LIN {X 0,Y 220.95,Z 365.337,A -85,B 0,C 180,E1 -21122.312,E2 -21122.312} C_VEL
LIN {X 0,Y 219.711,Z 400.675,A -85,B 0,C 180,E1 -21123.481,E2 -21123.481} C_VEL
LIN {X 0,Y 218.85,Z 411.091,A -85,B 0,C 180,E1 -21124.077,E2 -21124.077} C_VEL
LIN {X 0,Y 217.457,Z 422.982,A -85,B 0,C 180,E1 -21125.157,E2 -21125.157} C_VEL
LIN {X 0,Y 216.121,Z 431.792,A -85,B 0,C 180,E1 -21126.271,E2 -21126.271} C_VEL
LIN {X 0,Y 214.526,Z 440.18,A -85,B 0,C 180,E1 -21127.615,E2 -21127.615} C_VEL
LIN {X 0,Y 212.777,Z 448.104,A -85,B 0,C 180,E1 -21129.203,E2 -21129.203} C_VEL
LIN {X 0,Y 210.956,Z 455.495,A -85,B 0,C 180,E1 -21131.046,E2 -21131.046} C_VEL
LIN {X 0,Y 209.085,Z 462.983,A -85,B 0,C 180,E1 -21133.399,E2 -21133.399} C_VEL
LIN {X 0,Y 207.25,Z 469.848,A -85,B 0,C 180,E1 -21136.269,E2 -21136.269} C_VEL
LIN {X 0,Y 205.923,Z 475.039,A -85,B 0,C 180,E1 -21139.181,E2 -21139.181} C_VEL
LIN {X 0,Y 205.254,Z 477.703,A -85,B 0,C 180,E1 -21141.137,E2 -21141.137} C_VEL
LIN {X 0,Y 204.593,Z 480.62,A -85,B 0,C 180,E1 -21144.085,E2 -21144.085} C_VEL
LIN {X 0,Y 204.405,Z 481.892,A -85,B 0,C 180,E1 -21146.057,E2 -21146.057} C_VEL
LIN {X 0,Y 204.322,Z 482.694,A -85,B 0,C 180,E1 -21148.029,E2 -21148.029} C_VEL
LIN {X 0,Y 204.302,Z 482.999,A -85,B 0,C 180,E1 -21150,E2 -21150} C_VEL
LIN {X 0,Y 204.315,Z 482.717,A -85,B 0,C 180,E1 -21151.971,E2 -21151.971} C_VEL
LIN {X 0,Y 204.439,Z 481.698,A -85,B 0,C 180,E1 -21154.487,E2 -21154.487} C_VEL
LIN {X 0,Y 204.992,Z 479.021,A -85,B 0,C 180,E1 -21157.882,E2 -21157.882} C_VEL
LIN {X 0,Y 205.895,Z 475.26,A -85,B 0,C 180,E1 -21160.82,E2 -21160.82} C_VEL
LIN {X 0,Y 207.184,Z 470.127,A -85,B 0,C 180,E1 -21163.736,E2 -21163.736} C_VEL
LIN {X 0,Y 208.712,Z 464.607,A -85,B 0,C 180,E1 -21166.129,E2 -21166.129} C_VEL
LIN {X 0,Y 210.499,Z 457.67,A -85,B 0,C 180,E1 -21168.492,E2 -21168.492} C_VEL
LIN {X 0,Y 212.455,Z 449.707,A -85,B 0,C 180,E1 -21170.577,E2 -21170.577} C_VEL
LIN {X 0,Y 214.197,Z 442.115,A -85,B 0,C 180,E1 -21172.168,E2 -21172.168} C_VEL
LIN {X 0,Y 215.813,Z 434.156,A -85,B 0,C 180,E1 -21173.51,E2 -21173.51} C_VEL
LIN {X 0,Y 216.859,Z 427.803,A -85,B 0,C 180,E1 -21174.406,E2 -21174.406} C_VEL
LIN {X 0,Y 218.133,Z 418.906,A -85,B 0,C 180,E1 -21175.386,E2 -21175.386} C_VEL
LIN {X 0,Y 219.062,Z 409.592,A -85,B 0,C 180,E1 -21176.159,E2 -21176.159} C_VEL
LIN {X 0,Y 219.757,Z 400.653,A -85,B 0,C 180,E1 -21176.661,E2 -21176.661} C_VEL
LIN {X 0,Y 221.039,Z 365.121,A -85,B 0,C 180,E1 -21177.832,E2 -21177.832} C_VEL
LIN {X 0,Y 218.467,Z 349.485,A -85,B 0,C 180,E1 -21178.761,E2 -21178.761} C_VEL
LIN {X 0,Y 212.436,Z 334.283,A -85,B 0,C 180,E1 -21180.238,E2 -21180.238} C_VEL
LIN {X 0,Y 207.752,Z 323.941,A -85,B 0,C 180,E1 -21181.473,E2 -21181.473} C_VEL
LIN {X 0,Y 207.162,Z 321.361,A -85,B 0,C 180,E1 -21182.874,E2 -21182.874} C_VEL
LIN {X 0,Y 206.738,Z 319.61,A -85,B 0,C 180,E1 -21184.118,E2 -21184.118} C_VEL
LIN {X 0,Y 206.671,Z 319.549,A -85,B 0,C 180,E1 -21188.543,E2 -21188.543} C_VEL
LIN {X 0,Y 206.616,Z 319.531,A -85,B 0,C 180,E1 -21192.866,E2 -21192.866} C_VEL
LIN {X 0,Y 206.615,Z 319.554,A -85,B 0,C 180,E1 -21197.133,E2 -21197.133} C_VEL
LIN {X 0,Y 206.659,Z 319.506,A -85,B 0,C 180,E1 -21202.255,E2 -21202.255} C_VEL
LIN {X 0,Y 206.697,Z 319.538,A -85,B 0,C 180,E1 -21204.688,E2 -21204.688} C_VEL
LIN {X 0,Y 206.691,Z 319.539,A -85,B 0,C 180,E1 -21209.333,E2 -21209.333} C_VEL
LIN {X 0,Y 206.682,Z 319.552,A -85,B 0,C 180,E1 -21213.765,E2 -21213.765} C_VEL
LIN {X 0,Y 206.707,Z 319.528,A -85,B 0,C 180,E1 -21218.037,E2 -21218.037} C_VEL
LIN {X 0,Y 206.799,Z 319.538,A -85,B 0,C 180,E1 -21222.19,E2 -21222.19} C_VEL
LIN {X 0,Y 206.846,Z 319.508,A -85,B 0,C 180,E1 -21226.241,E2 -21226.241} C_VEL
LIN {X 0,Y 207.073,Z 319.503,A -85,B 0,C 180,E1 -21230.229,E2 -21230.229} C_VEL
LIN {X 0,Y 207.03,Z 319.487,A -85,B 0,C 180,E1 -21234.155,E2 -21234.155} C_VEL
LIN {X 0,Y 207.336,Z 319.463,A -85,B 0,C 180,E1 -21238.057,E2 -21238.057} C_VEL
LIN {X 0,Y 207.473,Z 319.455,A -85,B 0,C 180,E1 -21240,E2 -21240} C_VEL
LIN {X 0,Y 207.333,Z 319.464,A -85,B 0,C 180,E1 -21241.942,E2 -21241.942} C_VEL
LIN {X 0,Y 207.111,Z 319.493,A -85,B 0,C 180,E1 -21247.801,E2 -21247.801} C_VEL
LIN {X 0,Y 206.896,Z 319.513,A -85,B 0,C 180,E1 -21251.76,E2 -21251.76} C_VEL
LIN {X 0,Y 206.794,Z 319.527,A -85,B 0,C 180,E1 -21255.776,E2 -21255.776} C_VEL
LIN {X 0,Y 206.705,Z 319.542,A -85,B 0,C 180,E1 -21259.877,E2 -21259.877} C_VEL
LIN {X 0,Y 206.716,Z 319.539,A -85,B 0,C 180,E1 -21264.078,E2 -21264.078} C_VEL
LIN {X 0,Y 206.682,Z 319.541,A -85,B 0,C 180,E1 -21268.428,E2 -21268.428} C_VEL
LIN {X 0,Y 206.69,Z 319.552,A -85,B 0,C 180,E1 -21272.959,E2 -21272.959} C_VEL
LIN {X 0,Y 206.662,Z 319.507,A -85,B 0,C 180,E1 -21277.743,E2 -21277.743} C_VEL
LIN {X 0,Y 206.627,Z 319.53,A -85,B 0,C 180,E1 -21281.559,E2 -21281.559} C_VEL
LIN {X 0,Y 206.626,Z 319.552,A -85,B 0,C 180,E1 -21285.584,E2 -21285.584} C_VEL
LIN {X 0,Y 206.644,Z 319.525,A -85,B 0,C 180,E1 -21289.746,E2 -21289.746} C_VEL
LIN {X 0,Y 206.697,Z 319.53,A -85,B 0,C 180,E1 -21294.689,E2 -21294.689} C_VEL
LIN {X 0,Y 206.763,Z 319.832,A -85,B 0,C 180,E1 -21296.18,E2 -21296.18} C_VEL
LIN {X 0,Y 207.225,Z 321.798,A -85,B 0,C 180,E1 -21297.441,E2 -21297.441} C_VEL
LIN {X 0,Y 207.769,Z 324.004,A -85,B 0,C 180,E1 -21298.251,E2 -21298.251} C_VEL
LIN {X 0,Y 208.558,Z 327.091,A -85,B 0,C 180,E1 -21298.81,E2 -21298.81} C_VEL
LIN {X 0,Y 209.749,Z 332.596,A -85,B 0,C 180,E1 -21299.313,E2 -21299.313} C_VEL
LIN {X 0,Y 211.186,Z 347.134,A -85,B 0,C 180,E1 -21300.1,E2 -21300.1} C_VEL
LIN {X 0,Y 212.232,Z 351.094,A -85,B 0,C 180,E1 -21300.418,E2 -21300.418} C_VEL
LIN {X 0,Y 213.675,Z 358.475,A -85,B 0,C 180,E1 -21300.917,E2 -21300.917} C_VEL
LIN {X 0,Y 214.812,Z 367.699,A -85,B 0,C 180,E1 -21301.43,E2 -21301.43} C_VEL
LIN {X 0,Y 213.518,Z 400.025,A -85,B 0,C 180,E1 -21302.509,E2 -21302.509} C_VEL
LIN {X 0,Y 212.78,Z 409.431,A -85,B 0,C 180,E1 -21303.041,E2 -21303.041} C_VEL
LIN {X 0,Y 211.677,Z 418.832,A -85,B 0,C 180,E1 -21303.82,E2 -21303.82} C_VEL
LIN {X 0,Y 210.186,Z 429.315,A -85,B 0,C 180,E1 -21305.031,E2 -21305.031} C_VEL
LIN {X 0,Y 208.163,Z 439.443,A -85,B 0,C 180,E1 -21306.628,E2 -21306.628} C_VEL
LIN {X 0,Y 206.357,Z 447.487,A -85,B 0,C 180,E1 -21308.262,E2 -21308.262} C_VEL
LIN {X 0,Y 204.685,Z 454.131,A -85,B 0,C 180,E1 -21309.919,E2 -21309.919} C_VEL
LIN {X 0,Y 202.959,Z 460.438,A -85,B 0,C 180,E1 -21311.842,E2 -21311.842} C_VEL
LIN {X 0,Y 201.558,Z 465.676,A -85,B 0,C 180,E1 -21313.803,E2 -21313.803} C_VEL
LIN {X 0,Y 200.308,Z 470.043,A -85,B 0,C 180,E1 -21315.783,E2 -21315.783} C_VEL
LIN {X 0,Y 198.917,Z 475.192,A -85,B 0,C 180,E1 -21318.795,E2 -21318.795} C_VEL
LIN {X 0,Y 197.976,Z 478.97,A -85,B 0,C 180,E1 -21321.837,E2 -21321.837} C_VEL
LIN {X 0,Y 197.59,Z 480.702,A -85,B 0,C 180,E1 -21323.875,E2 -21323.875} C_VEL
LIN {X 0,Y 197.332,Z 481.941,A -85,B 0,C 180,E1 -21325.915,E2 -21325.915} C_VEL
LIN {X 0,Y 197.234,Z 482.71,A -85,B 0,C 180,E1 -21327.958,E2 -21327.958} C_VEL
LIN {X 0,Y 197.21,Z 483,A -85,B 0,C 180,E1 -21330,E2 -21330} C_VEL
LIN {X 0,Y 197.232,Z 482.701,A -85,B 0,C 180,E1 -21332.042,E2 -21332.042} C_VEL
LIN {X 0,Y 197.336,Z 481.816,A -85,B 0,C 180,E1 -21334.291,E2 -21334.291} C_VEL
LIN {X 0,Y 197.523,Z 480.656,A -85,B 0,C 180,E1 -21336.127,E2 -21336.127} C_VEL
LIN {X 0,Y 198.238,Z 477.754,A -85,B 0,C 180,E1 -21339.18,E2 -21339.18} C_VEL
LIN {X 0,Y 198.911,Z 475.107,A -85,B 0,C 180,E1 -21341.205,E2 -21341.205} C_VEL
LIN {X 0,Y 200.301,Z 469.932,A -85,B 0,C 180,E1 -21344.218,E2 -21344.218} C_VEL
LIN {X 0,Y 202.263,Z 463.105,A -85,B 0,C 180,E1 -21347.178,E2 -21347.178} C_VEL
LIN {X 0,Y 204.226,Z 455.644,A -85,B 0,C 180,E1 -21349.604,E2 -21349.604} C_VEL
LIN {X 0,Y 206.112,Z 448.282,A -85,B 0,C 180,E1 -21351.503,E2 -21351.503} C_VEL
LIN {X 0,Y 207.939,Z 440.395,A -85,B 0,C 180,E1 -21353.135,E2 -21353.135} C_VEL
LIN {X 0,Y 209.55,Z 432.053,A -85,B 0,C 180,E1 -21354.521,E2 -21354.521} C_VEL
LIN {X 0,Y 211.157,Z 422.131,A -85,B 0,C 180,E1 -21355.803,E2 -21355.803} C_VEL
LIN {X 0,Y 212.607,Z 410.515,A -85,B 0,C 180,E1 -21356.836,E2 -21356.836} C_VEL
LIN {X 0,Y 213.421,Z 400.836,A -85,B 0,C 180,E1 -21357.402,E2 -21357.402} C_VEL
LIN {X 0,Y 214.677,Z 366.325,A -85,B 0,C 180,E1 -21358.58,E2 -21358.58} C_VEL
LIN {X 0,Y 212.372,Z 351.475,A -85,B 0,C 180,E1 -21359.482,E2 -21359.482} C_VEL
LIN {X 0,Y 206.305,Z 336.552,A -85,B 0,C 180,E1 -21361.03,E2 -21361.03} C_VEL
LIN {X 0,Y 200.492,Z 323.95,A -85,B 0,C 180,E1 -21362.63,E2 -21362.63} C_VEL
LIN {X 0,Y 199.816,Z 321.165,A -85,B 0,C 180,E1 -21364.246,E2 -21364.246} C_VEL
LIN {X 0,Y 199.669,Z 320.48,A -85,B 0,C 180,E1 -21364.845,E2 -21364.845} C_VEL
LIN {X 0,Y 199.593,Z 320.412,A -85,B 0,C 180,E1 -21369.331,E2 -21369.331} C_VEL
LIN {X 0,Y 199.562,Z 320.404,A -85,B 0,C 180,E1 -21372.306,E2 -21372.306} C_VEL
LIN {X 0,Y 199.572,Z 320.438,A -85,B 0,C 180,E1 -21375.227,E2 -21375.227} C_VEL
LIN {X 0,Y 199.566,Z 320.413,A -85,B 0,C 180,E1 -21378.002,E2 -21378.002} C_VEL
LIN {X 0,Y 199.593,Z 320.378,A -85,B 0,C 180,E1 -21380.772,E2 -21380.772} C_VEL
LIN {X 0,Y 199.607,Z 320.432,A -85,B 0,C 180,E1 -21385.713,E2 -21385.713} C_VEL
LIN {X 0,Y 199.681,Z 320.42,A -85,B 0,C 180,E1 -21388.134,E2 -21388.134} C_VEL
LIN {X 0,Y 199.63,Z 320.428,A -85,B 0,C 180,E1 -21392.764,E2 -21392.764} C_VEL
LIN {X 0,Y 199.666,Z 320.405,A -85,B 0,C 180,E1 -21397.221,E2 -21397.221} C_VEL
LIN {X 0,Y 199.741,Z 320.416,A -85,B 0,C 180,E1 -21401.803,E2 -21401.803} C_VEL
LIN {X 0,Y 199.763,Z 320.39,A -85,B 0,C 180,E1 -21405.743,E2 -21405.743} C_VEL
LIN {X 0,Y 200.019,Z 320.379,A -85,B 0,C 180,E1 -21409.882,E2 -21409.882} C_VEL
LIN {X 0,Y 199.994,Z 320.363,A -85,B 0,C 180,E1 -21413.949,E2 -21413.949} C_VEL
LIN {X 0,Y 200.278,Z 320.342,A -85,B 0,C 180,E1 -21417.989,E2 -21417.989} C_VEL
LIN {X 0,Y 200.44,Z 320.331,A -85,B 0,C 180,E1 -21420,E2 -21420} C_VEL
LIN {X 0,Y 199.973,Z 320.362,A -85,B 0,C 180,E1 -21424.031,E2 -21424.031} C_VEL
LIN {X 0,Y 200.06,Z 320.373,A -85,B 0,C 180,E1 -21428.078,E2 -21428.078} C_VEL
LIN {X 0,Y 199.846,Z 320.388,A -85,B 0,C 180,E1 -21432.181,E2 -21432.181} C_VEL
LIN {X 0,Y 199.735,Z 320.41,A -85,B 0,C 180,E1 -21436.35,E2 -21436.35} C_VEL
LIN {X 0,Y 199.639,Z 320.417,A -85,B 0,C 180,E1 -21440.612,E2 -21440.612} C_VEL
LIN {X 0,Y 199.631,Z 320.427,A -85,B 0,C 180,E1 -21444.99,E2 -21444.99} C_VEL
LIN {X 0,Y 199.604,Z 320.416,A -85,B 0,C 180,E1 -21449.534,E2 -21449.534} C_VEL
LIN {X 0,Y 199.662,Z 320.425,A -85,B 0,C 180,E1 -21452.353,E2 -21452.353} C_VEL
LIN {X 0,Y 199.613,Z 320.397,A -85,B 0,C 180,E1 -21456.765,E2 -21456.765} C_VEL
LIN {X 0,Y 199.591,Z 320.379,A -85,B 0,C 180,E1 -21459.332,E2 -21459.332} C_VEL
LIN {X 0,Y 199.563,Z 320.418,A -85,B 0,C 180,E1 -21462.308,E2 -21462.308} C_VEL
LIN {X 0,Y 199.573,Z 320.435,A -85,B 0,C 180,E1 -21465.228,E2 -21465.228} C_VEL
LIN {X 0,Y 199.567,Z 320.401,A -85,B 0,C 180,E1 -21468.003,E2 -21468.003} C_VEL
LIN {X 0,Y 199.596,Z 320.412,A -85,B 0,C 180,E1 -21470.773,E2 -21470.773} C_VEL
LIN {X 0,Y 199.728,Z 320.655,A -85,B 0,C 180,E1 -21475.453,E2 -21475.453} C_VEL
LIN {X 0,Y 200.467,Z 323.816,A -85,B 0,C 180,E1 -21477.38,E2 -21477.38} C_VEL
LIN {X 0,Y 202.785,Z 329.044,A -85,B 0,C 180,E1 -21478.109,E2 -21478.109} C_VEL
LIN {X 0,Y 208.66,Z 342.11,A -85,B 0,C 180,E1 -21479.62,E2 -21479.62} C_VEL
LIN {X 0,Y 212.507,Z 352.019,A -85,B 0,C 180,E1 -21480.604,E2 -21480.604} C_VEL
LIN {X 0,Y 214.697,Z 366.722,A -85,B 0,C 180,E1 -21481.483,E2 -21481.483} C_VEL
LIN {X 0,Y 213.422,Z 400.147,A -85,B 0,C 180,E1 -21482.608,E2 -21482.608} C_VEL
LIN {X 0,Y 212.631,Z 409.776,A -85,B 0,C 180,E1 -21483.153,E2 -21483.153} C_VEL
LIN {X 0,Y 211.516,Z 419.764,A -85,B 0,C 180,E1 -21484.006,E2 -21484.006} C_VEL
LIN {X 0,Y 209.91,Z 430.293,A -85,B 0,C 180,E1 -21485.26,E2 -21485.26} C_VEL
LIN {X 0,Y 207.983,Z 440.184,A -85,B 0,C 180,E1 -21486.87,E2 -21486.87} C_VEL
LIN {X 0,Y 206.16,Z 448.107,A -85,B 0,C 180,E1 -21488.503,E2 -21488.503} C_VEL
LIN {X 0,Y 204.262,Z 455.497,A -85,B 0,C 180,E1 -21490.4,E2 -21490.4} C_VEL
LIN {X 0,Y 202.29,Z 462.985,A -85,B 0,C 180,E1 -21492.824,E2 -21492.824} C_VEL
LIN {X 0,Y 200.342,Z 469.849,A -85,B 0,C 180,E1 -21495.785,E2 -21495.785} C_VEL
LIN {X 0,Y 198.94,Z 475.04,A -85,B 0,C 180,E1 -21498.796,E2 -21498.796} C_VEL
LIN {X 0,Y 198.242,Z 477.703,A -85,B 0,C 180,E1 -21500.82,E2 -21500.82} C_VEL
LIN {X 0,Y 197.525,Z 480.621,A -85,B 0,C 180,E1 -21503.873,E2 -21503.873} C_VEL
LIN {X 0,Y 197.326,Z 481.893,A -85,B 0,C 180,E1 -21505.915,E2 -21505.915} C_VEL
LIN {X 0,Y 197.234,Z 482.694,A -85,B 0,C 180,E1 -21507.958,E2 -21507.958} C_VEL
LIN {X 0,Y 197.211,Z 482.999,A -85,B 0,C 180,E1 -21510,E2 -21510} C_VEL
LIN {X 0,Y 197.228,Z 482.717,A -85,B 0,C 180,E1 -21512.042,E2 -21512.042} C_VEL
LIN {X 0,Y 197.338,Z 481.865,A -85,B 0,C 180,E1 -21514.291,E2 -21514.291} C_VEL
LIN {X 0,Y 197.525,Z 480.738,A -85,B 0,C 180,E1 -21516.127,E2 -21516.127} C_VEL
LIN {X 0,Y 198.239,Z 477.869,A -85,B 0,C 180,E1 -21519.18,E2 -21519.18} C_VEL
LIN {X 0,Y 198.907,Z 475.258,A -85,B 0,C 180,E1 -21521.205,E2 -21521.205} C_VEL
LIN {X 0,Y 200.282,Z 470.126,A -85,B 0,C 180,E1 -21524.219,E2 -21524.219} C_VEL
LIN {X 0,Y 201.894,Z 464.605,A -85,B 0,C 180,E1 -21526.689,E2 -21526.689} C_VEL
LIN {X 0,Y 203.756,Z 457.667,A -85,B 0,C 180,E1 -21529.127,E2 -21529.127} C_VEL
LIN {X 0,Y 205.831,Z 449.703,A -85,B 0,C 180,E1 -21531.271,E2 -21531.271} C_VEL
LIN {X 0,Y 207.639,Z 442.111,A -85,B 0,C 180,E1 -21532.907,E2 -21532.907} C_VEL
LIN {X 0,Y 209.328,Z 434.151,A -85,B 0,C 180,E1 -21534.285,E2 -21534.285} C_VEL
LIN {X 0,Y 210.745,Z 425.924,A -85,B 0,C 180,E1 -21535.426,E2 -21535.426} C_VEL
LIN {X 0,Y 211.861,Z 417.634,A -85,B 0,C 180,E1 -21536.332,E2 -21536.332} C_VEL
LIN {X 0,Y 212.757,Z 409.338,A -85,B 0,C 180,E1 -21537.015,E2 -21537.015} C_VEL
LIN {X 0,Y 213.439,Z 400.806,A -85,B 0,C 180,E1 -21537.507,E2 -21537.507} C_VEL
LIN {X 0,Y 214.789,Z 366.132,A -85,B 0,C 180,E1 -21538.677,E2 -21538.677} C_VEL
LIN {X 0,Y 212.416,Z 351.696,A -85,B 0,C 180,E1 -21539.576,E2 -21539.576} C_VEL
LIN {X 0,Y 206.152,Z 336.12,A -85,B 0,C 180,E1 -21541.187,E2 -21541.187} C_VEL
LIN {X 0,Y 200.525,Z 323.991,A -85,B 0,C 180,E1 -21542.737,E2 -21542.737} C_VEL
LIN {X 0,Y 200.187,Z 322.632,A -85,B 0,C 180,E1 -21543.385,E2 -21543.385} C_VEL
LIN {X 0,Y 199.67,Z 320.525,A -85,B 0,C 180,E1 -21544.844,E2 -21544.844} C_VEL
LIN {X 0,Y 199.593,Z 320.414,A -85,B 0,C 180,E1 -21549.331,E2 -21549.331} C_VEL
LIN {X 0,Y 199.563,Z 320.403,A -85,B 0,C 180,E1 -21552.306,E2 -21552.306} C_VEL
LIN {X 0,Y 199.573,Z 320.437,A -85,B 0,C 180,E1 -21555.226,E2 -21555.226} C_VEL
LIN {X 0,Y 199.566,Z 320.416,A -85,B 0,C 180,E1 -21558.001,E2 -21558.001} C_VEL
LIN {X 0,Y 199.59,Z 320.379,A -85,B 0,C 180,E1 -21560.773,E2 -21560.773} C_VEL
LIN {X 0,Y 199.608,Z 320.43,A -85,B 0,C 180,E1 -21565.712,E2 -21565.712} C_VEL
LIN {X 0,Y 199.682,Z 320.421,A -85,B 0,C 180,E1 -21568.133,E2 -21568.133} C_VEL
LIN {X 0,Y 199.631,Z 320.427,A -85,B 0,C 180,E1 -21572.763,E2 -21572.763} C_VEL
LIN {X 0,Y 199.666,Z 320.406,A -85,B 0,C 180,E1 -21577.22,E2 -21577.22} C_VEL
LIN {X 0,Y 199.742,Z 320.416,A -85,B 0,C 180,E1 -21581.802,E2 -21581.802} C_VEL
LIN {X 0,Y 199.763,Z 320.39,A -85,B 0,C 180,E1 -21585.743,E2 -21585.743} C_VEL
LIN {X 0,Y 200.019,Z 320.379,A -85,B 0,C 180,E1 -21589.881,E2 -21589.881} C_VEL
LIN {X 0,Y 199.994,Z 320.364,A -85,B 0,C 180,E1 -21593.948,E2 -21593.948} C_VEL
LIN {X 0,Y 200.278,Z 320.341,A -85,B 0,C 180,E1 -21597.989,E2 -21597.989} C_VEL
LIN {X 0,Y 200.44,Z 320.331,A -85,B 0,C 180,E1 -21600,E2 -21600} C_VEL
LIN {X 0,Y 199.972,Z 320.362,A -85,B 0,C 180,E1 -21604.03,E2 -21604.03} C_VEL
LIN {X 0,Y 200.06,Z 320.373,A -85,B 0,C 180,E1 -21608.078,E2 -21608.078} C_VEL
LIN {X 0,Y 199.846,Z 320.388,A -85,B 0,C 180,E1 -21612.181,E2 -21612.181} C_VEL
LIN {X 0,Y 199.735,Z 320.411,A -85,B 0,C 180,E1 -21616.349,E2 -21616.349} C_VEL
LIN {X 0,Y 199.638,Z 320.416,A -85,B 0,C 180,E1 -21620.612,E2 -21620.612} C_VEL
LIN {X 0,Y 199.631,Z 320.427,A -85,B 0,C 180,E1 -21624.99,E2 -21624.99} C_VEL
LIN {X 0,Y 199.603,Z 320.416,A -85,B 0,C 180,E1 -21629.534,E2 -21629.534} C_VEL
LIN {X 0,Y 199.661,Z 320.426,A -85,B 0,C 180,E1 -21632.353,E2 -21632.353} C_VEL
LIN {X 0,Y 199.612,Z 320.395,A -85,B 0,C 180,E1 -21636.765,E2 -21636.765} C_VEL
LIN {X 0,Y 199.59,Z 320.379,A -85,B 0,C 180,E1 -21639.332,E2 -21639.332} C_VEL
LIN {X 0,Y 199.562,Z 320.421,A -85,B 0,C 180,E1 -21642.308,E2 -21642.308} C_VEL
LIN {X 0,Y 199.572,Z 320.434,A -85,B 0,C 180,E1 -21645.228,E2 -21645.228} C_VEL
LIN {X 0,Y 199.566,Z 320.401,A -85,B 0,C 180,E1 -21648.003,E2 -21648.003} C_VEL
LIN {X 0,Y 199.594,Z 320.415,A -85,B 0,C 180,E1 -21650.773,E2 -21650.773} C_VEL
LIN {X 0,Y 199.713,Z 320.637,A -85,B 0,C 180,E1 -21655.307,E2 -21655.307} C_VEL
LIN {X 0,Y 200.423,Z 323.64,A -85,B 0,C 180,E1 -21657.208,E2 -21657.208} C_VEL
LIN {X 0,Y 201.812,Z 326.976,A -85,B 0,C 180,E1 -21657.734,E2 -21657.734} C_VEL
LIN {X 0,Y 207.532,Z 339.186,A -85,B 0,C 180,E1 -21659.21,E2 -21659.21} C_VEL
LIN {X 0,Y 212.232,Z 351.094,A -85,B 0,C 180,E1 -21660.418,E2 -21660.418} C_VEL
LIN {X 0,Y 213.046,Z 354.757,A -85,B 0,C 180,E1 -21660.681,E2 -21660.681} C_VEL
LIN {X 0,Y 212.87,Z 360.592,A -85,B 0,C 180,E1 -21660.876,E2 -21660.876} C_VEL
LIN {X 0,Y 211.652,Z 366.44,A -85,B 0,C 180,E1 -21660.915,E2 -21660.915} C_VEL
LIN {X 0,Y 208.505,Z 378.509,A -85,B 0,C 180,E1 -21660.899,E2 -21660.899} C_VEL
LIN {X 0,Y 208.016,Z 382.602,A -85,B 0,C 180,E1 -21660.983,E2 -21660.983} C_VEL
LIN {X 0,Y 207.142,Z 402.34,A -85,B 0,C 180,E1 -21661.71,E2 -21661.71} C_VEL
LIN {X 0,Y 206.016,Z 413.671,A -85,B 0,C 180,E1 -21662.456,E2 -21662.456} C_VEL
LIN {X 0,Y 204.623,Z 423.738,A -85,B 0,C 180,E1 -21663.481,E2 -21663.481} C_VEL
LIN {X 0,Y 203.157,Z 432.399,A -85,B 0,C 180,E1 -21664.654,E2 -21664.654} C_VEL
LIN {X 0,Y 201.412,Z 440.676,A -85,B 0,C 180,E1 -21666.069,E2 -21666.069} C_VEL
LIN {X 0,Y 199.515,Z 448.511,A -85,B 0,C 180,E1 -21667.749,E2 -21667.749} C_VEL
LIN {X 0,Y 197.557,Z 455.837,A -85,B 0,C 180,E1 -21669.706,E2 -21669.706} C_VEL
LIN {X 0,Y 195.486,Z 463.268,A -85,B 0,C 180,E1 -21672.207,E2 -21672.207} C_VEL
LIN {X 0,Y 193.42,Z 470.044,A -85,B 0,C 180,E1 -21675.265,E2 -21675.265} C_VEL
LIN {X 0,Y 191.951,Z 475.193,A -85,B 0,C 180,E1 -21678.383,E2 -21678.383} C_VEL
LIN {X 0,Y 190.955,Z 478.971,A -85,B 0,C 180,E1 -21681.534,E2 -21681.534} C_VEL
LIN {X 0,Y 190.528,Z 480.703,A -85,B 0,C 180,E1 -21683.647,E2 -21683.647} C_VEL
LIN {X 0,Y 190.222,Z 482.043,A -85,B 0,C 180,E1 -21685.985,E2 -21685.985} C_VEL
LIN {X 0,Y 190.149,Z 482.71,A -85,B 0,C 180,E1 -21687.882,E2 -21687.882} C_VEL
LIN {X 0,Y 190.121,Z 483,A -85,B 0,C 180,E1 -21690,E2 -21690} C_VEL
LIN {X 0,Y 190.147,Z 482.701,A -85,B 0,C 180,E1 -21692.118,E2 -21692.118} C_VEL
LIN {X 0,Y 190.238,Z 481.914,A -85,B 0,C 180,E1 -21694.237,E2 -21694.237} C_VEL
LIN {X 0,Y 190.468,Z 480.656,A -85,B 0,C 180,E1 -21696.355,E2 -21696.355} C_VEL
LIN {X 0,Y 191.226,Z 477.753,A -85,B 0,C 180,E1 -21699.519,E2 -21699.519} C_VEL
LIN {X 0,Y 191.945,Z 475.105,A -85,B 0,C 180,E1 -21701.617,E2 -21701.617} C_VEL
LIN {X 0,Y 193.411,Z 469.931,A -85,B 0,C 180,E1 -21704.735,E2 -21704.735} C_VEL
LIN {X 0,Y 195.484,Z 463.103,A -85,B 0,C 180,E1 -21707.793,E2 -21707.793} C_VEL
LIN {X 0,Y 197.566,Z 455.641,A -85,B 0,C 180,E1 -21710.293,E2 -21710.293} C_VEL
LIN {X 0,Y 199.507,Z 448.279,A -85,B 0,C 180,E1 -21712.252,E2 -21712.252} C_VEL
LIN {X 0,Y 201.436,Z 440.391,A -85,B 0,C 180,E1 -21713.928,E2 -21713.928} C_VEL
LIN {X 0,Y 203.107,Z 432.048,A -85,B 0,C 180,E1 -21715.353,E2 -21715.353} C_VEL
LIN {X 0,Y 204.795,Z 422.129,A -85,B 0,C 180,E1 -21716.666,E2 -21716.666} C_VEL
LIN {X 0,Y 206.295,Z 410.586,A -85,B 0,C 180,E1 -21717.72,E2 -21717.72} C_VEL
LIN {X 0,Y 207.148,Z 401.037,A -85,B 0,C 180,E1 -21718.294,E2 -21718.294} C_VEL
LIN {X 0,Y 208.414,Z 367.129,A -85,B 0,C 180,E1 -21719.49,E2 -21719.49} C_VEL
LIN {X 0,Y 206.398,Z 353.934,A -85,B 0,C 180,E1 -21720.326,E2 -21720.326} C_VEL
LIN {X 0,Y 200.763,Z 339.948,A -85,B 0,C 180,E1 -21721.846,E2 -21721.846} C_VEL
LIN {X 0,Y 194.681,Z 327.042,A -85,B 0,C 180,E1 -21723.521,E2 -21723.521} C_VEL
LIN {X 0,Y 193.198,Z 323.808,A -85,B 0,C 180,E1 -21724.063,E2 -21724.063} C_VEL
LIN {X 0,Y 192.591,Z 321.4,A -85,B 0,C 180,E1 -21725.635,E2 -21725.635} C_VEL
LIN {X 0,Y 192.502,Z 321.285,A -85,B 0,C 180,E1 -21729.944,E2 -21729.944} C_VEL
LIN {X 0,Y 192.483,Z 321.305,A -85,B 0,C 180,E1 -21733.925,E2 -21733.925} C_VEL
LIN {X 0,Y 192.5,Z 321.273,A -85,B 0,C 180,E1 -21738.916,E2 -21738.916} C_VEL
LIN {X 0,Y 192.578,Z 321.272,A -85,B 0,C 180,E1 -21743.404,E2 -21743.404} C_VEL
LIN {X 0,Y 192.601,Z 321.307,A -85,B 0,C 180,E1 -21747.061,E2 -21747.061} C_VEL
LIN {X 0,Y 192.615,Z 321.293,A -85,B 0,C 180,E1 -21751.684,E2 -21751.684} C_VEL
LIN {X 0,Y 192.657,Z 321.283,A -85,B 0,C 180,E1 -21756.343,E2 -21756.343} C_VEL
LIN {X 0,Y 192.69,Z 321.294,A -85,B 0,C 180,E1 -21761.492,E2 -21761.492} C_VEL
LIN {X 0,Y 192.768,Z 321.264,A -85,B 0,C 180,E1 -21767.365,E2 -21767.365} C_VEL
LIN {X 0,Y 193.02,Z 321.253,A -85,B 0,C 180,E1 -21771.626,E2 -21771.626} C_VEL
LIN {X 0,Y 193.222,Z 321.22,A -85,B 0,C 180,E1 -21777.916,E2 -21777.916} C_VEL
LIN {X 0,Y 193.407,Z 321.208,A -85,B 0,C 180,E1 -21780,E2 -21780} C_VEL
LIN {X 0,Y 192.92,Z 321.238,A -85,B 0,C 180,E1 -21784.178,E2 -21784.178} C_VEL
LIN {X 0,Y 193.013,Z 321.253,A -85,B 0,C 180,E1 -21788.375,E2 -21788.375} C_VEL
LIN {X 0,Y 192.768,Z 321.264,A -85,B 0,C 180,E1 -21792.636,E2 -21792.636} C_VEL
LIN {X 0,Y 192.69,Z 321.294,A -85,B 0,C 180,E1 -21798.509,E2 -21798.509} C_VEL
LIN {X 0,Y 192.622,Z 321.293,A -85,B 0,C 180,E1 -21804.199,E2 -21804.199} C_VEL
LIN {X 0,Y 192.597,Z 321.291,A -85,B 0,C 180,E1 -21808.865,E2 -21808.865} C_VEL
LIN {X 0,Y 192.592,Z 321.309,A -85,B 0,C 180,E1 -21813.187,E2 -21813.187} C_VEL
LIN {X 0,Y 192.538,Z 321.257,A -85,B 0,C 180,E1 -21818.355,E2 -21818.355} C_VEL
LIN {X 0,Y 192.483,Z 321.313,A -85,B 0,C 180,E1 -21823.094,E2 -21823.094} C_VEL
LIN {X 0,Y 192.481,Z 321.292,A -85,B 0,C 180,E1 -21826.908,E2 -21826.908} C_VEL
LIN {X 0,Y 192.542,Z 321.305,A -85,B 0,C 180,E1 -21831.647,E2 -21831.647} C_VEL
LIN {X 0,Y 192.603,Z 321.428,A -85,B 0,C 180,E1 -21834.455,E2 -21834.455} C_VEL
LIN {X 0,Y 193.177,Z 323.727,A -85,B 0,C 180,E1 -21835.955,E2 -21835.955} C_VEL
LIN {X 0,Y 194.949,Z 327.476,A -85,B 0,C 180,E1 -21836.595,E2 -21836.595} C_VEL
LIN {X 0,Y 202.401,Z 343.758,A -85,B 0,C 180,E1 -21838.642,E2 -21838.642} C_VEL
LIN {X 0,Y 206.582,Z 354.443,A -85,B 0,C 180,E1 -21839.769,E2 -21839.769} C_VEL
LIN {X 0,Y 208.417,Z 366.668,A -85,B 0,C 180,E1 -21840.538,E2 -21840.538} C_VEL
LIN {X 0,Y 207.163,Z 400.025,A -85,B 0,C 180,E1 -21841.699,E2 -21841.699} C_VEL
LIN {X 0,Y 206.297,Z 410.087,A -85,B 0,C 180,E1 -21842.284,E2 -21842.284} C_VEL
LIN {X 0,Y 204.949,Z 421.396,A -85,B 0,C 180,E1 -21843.301,E2 -21843.301} C_VEL
LIN {X 0,Y 203.186,Z 431.802,A -85,B 0,C 180,E1 -21844.657,E2 -21844.657} C_VEL
LIN {X 0,Y 201.47,Z 440.188,A -85,B 0,C 180,E1 -21846.077,E2 -21846.077} C_VEL
LIN {X 0,Y 199.552,Z 448.111,A -85,B 0,C 180,E1 -21847.753,E2 -21847.753} C_VEL
LIN {X 0,Y 198.083,Z 453.799,A -85,B 0,C 180,E1 -21849.219,E2 -21849.219} C_VEL
LIN {X 0,Y 196.26,Z 460.155,A -85,B 0,C 180,E1 -21851.199,E2 -21851.199} C_VEL
LIN {X 0,Y 194.763,Z 465.439,A -85,B 0,C 180,E1 -21853.222,E2 -21853.222} C_VEL
LIN {X 0,Y 193.452,Z 469.851,A -85,B 0,C 180,E1 -21855.268,E2 -21855.268} C_VEL
LIN {X 0,Y 191.976,Z 475.042,A -85,B 0,C 180,E1 -21858.384,E2 -21858.384} C_VEL
LIN {X 0,Y 191.23,Z 477.704,A -85,B 0,C 180,E1 -21860.481,E2 -21860.481} C_VEL
LIN {X 0,Y 190.47,Z 480.621,A -85,B 0,C 180,E1 -21863.645,E2 -21863.645} C_VEL
LIN {X 0,Y 190.219,Z 482.003,A -85,B 0,C 180,E1 -21866.005,E2 -21866.005} C_VEL
LIN {X 0,Y 190.149,Z 482.694,A -85,B 0,C 180,E1 -21867.882,E2 -21867.882} C_VEL
LIN {X 0,Y 190.122,Z 482.999,A -85,B 0,C 180,E1 -21870,E2 -21870} C_VEL
LIN {X 0,Y 190.142,Z 482.717,A -85,B 0,C 180,E1 -21872.118,E2 -21872.118} C_VEL
LIN {X 0,Y 190.24,Z 481.962,A -85,B 0,C 180,E1 -21874.237,E2 -21874.237} C_VEL
LIN {X 0,Y 190.47,Z 480.737,A -85,B 0,C 180,E1 -21876.355,E2 -21876.355} C_VEL
LIN {X 0,Y 191.227,Z 477.868,A -85,B 0,C 180,E1 -21879.519,E2 -21879.519} C_VEL
LIN {X 0,Y 191.94,Z 475.257,A -85,B 0,C 180,E1 -21881.618,E2 -21881.618} C_VEL
LIN {X 0,Y 193.405,Z 470.124,A -85,B 0,C 180,E1 -21884.736,E2 -21884.736} C_VEL
LIN {X 0,Y 195.102,Z 464.603,A -85,B 0,C 180,E1 -21887.288,E2 -21887.288} C_VEL
LIN {X 0,Y 197.055,Z 457.665,A -85,B 0,C 180,E1 -21889.804,E2 -21889.804} C_VEL
LIN {X 0,Y 199.226,Z 449.7,A -85,B 0,C 180,E1 -21892.012,E2 -21892.012} C_VEL
LIN {X 0,Y 201.121,Z 442.107,A -85,B 0,C 180,E1 -21893.694,E2 -21893.694} C_VEL
LIN {X 0,Y 202.878,Z 434.146,A -85,B 0,C 180,E1 -21895.109,E2 -21895.109} C_VEL
LIN {X 0,Y 204.373,Z 425.918,A -85,B 0,C 180,E1 -21896.279,E2 -21896.279} C_VEL
LIN {X 0,Y 205.553,Z 417.176,A -85,B 0,C 180,E1 -21897.257,E2 -21897.257} C_VEL
LIN {X 0,Y 206.579,Z 408.177,A -85,B 0,C 180,E1 -21897.987,E2 -21897.987} C_VEL
LIN {X 0,Y 207.265,Z 399.113,A -85,B 0,C 180,E1 -21898.489,E2 -21898.489} C_VEL
LIN {X 0,Y 208.517,Z 366.663,A -85,B 0,C 180,E1 -21899.603,E2 -21899.603} C_VEL
LIN {X 0,Y 206.489,Z 354.115,A -85,B 0,C 180,E1 -21900.417,E2 -21900.417} C_VEL
LIN {X 0,Y 200.117,Z 338.31,A -85,B 0,C 180,E1 -21902.147,E2 -21902.147} C_VEL
LIN {X 0,Y 194.526,Z 326.797,A -85,B 0,C 180,E1 -21903.685,E2 -21903.685} C_VEL
LIN {X 0,Y 193.162,Z 323.667,A -85,B 0,C 180,E1 -21904.233,E2 -21904.233} C_VEL
LIN {X 0,Y 192.595,Z 321.429,A -85,B 0,C 180,E1 -21905.721,E2 -21905.721} C_VEL
LIN {X 0,Y 192.503,Z 321.286,A -85,B 0,C 180,E1 -21909.943,E2 -21909.943} C_VEL
LIN {X 0,Y 192.483,Z 321.302,A -85,B 0,C 180,E1 -21913.925,E2 -21913.925} C_VEL
LIN {X 0,Y 192.499,Z 321.276,A -85,B 0,C 180,E1 -21918.916,E2 -21918.916} C_VEL
LIN {X 0,Y 192.577,Z 321.27,A -85,B 0,C 180,E1 -21923.404,E2 -21923.404} C_VEL
LIN {X 0,Y 192.602,Z 321.307,A -85,B 0,C 180,E1 -21927.06,E2 -21927.06} C_VEL
LIN {X 0,Y 192.615,Z 321.292,A -85,B 0,C 180,E1 -21931.684,E2 -21931.684} C_VEL
LIN {X 0,Y 192.658,Z 321.284,A -85,B 0,C 180,E1 -21936.342,E2 -21936.342} C_VEL
LIN {X 0,Y 192.69,Z 321.294,A -85,B 0,C 180,E1 -21941.491,E2 -21941.491} C_VEL
LIN {X 0,Y 192.769,Z 321.263,A -85,B 0,C 180,E1 -21947.364,E2 -21947.364} C_VEL
LIN {X 0,Y 193.02,Z 321.253,A -85,B 0,C 180,E1 -21951.625,E2 -21951.625} C_VEL
LIN {X 0,Y 193.222,Z 321.219,A -85,B 0,C 180,E1 -21957.915,E2 -21957.915} C_VEL
LIN {X 0,Y 193.407,Z 321.207,A -85,B 0,C 180,E1 -21960,E2 -21960} C_VEL
LIN {X 0,Y 192.92,Z 321.238,A -85,B 0,C 180,E1 -21964.178,E2 -21964.178} C_VEL
LIN {X 0,Y 193.013,Z 321.254,A -85,B 0,C 180,E1 -21968.375,E2 -21968.375} C_VEL
LIN {X 0,Y 192.768,Z 321.264,A -85,B 0,C 180,E1 -21972.635,E2 -21972.635} C_VEL
LIN {X 0,Y 192.69,Z 321.294,A -85,B 0,C 180,E1 -21978.508,E2 -21978.508} C_VEL
LIN {X 0,Y 192.621,Z 321.294,A -85,B 0,C 180,E1 -21984.199,E2 -21984.199} C_VEL
LIN {X 0,Y 192.596,Z 321.29,A -85,B 0,C 180,E1 -21988.865,E2 -21988.865} C_VEL
LIN {X 0,Y 192.591,Z 321.309,A -85,B 0,C 180,E1 -21993.187,E2 -21993.187} C_VEL
LIN {X 0,Y 192.537,Z 321.256,A -85,B 0,C 180,E1 -21998.355,E2 -21998.355} C_VEL
LIN {X 0,Y 192.482,Z 321.315,A -85,B 0,C 180,E1 -22003.094,E2 -22003.094} C_VEL
LIN {X 0,Y 192.48,Z 321.29,A -85,B 0,C 180,E1 -22006.908,E2 -22006.908} C_VEL
LIN {X 0,Y 192.539,Z 321.308,A -85,B 0,C 180,E1 -22011.646,E2 -22011.646} C_VEL
LIN {X 0,Y 192.611,Z 321.565,A -85,B 0,C 180,E1 -22014.455,E2 -22014.455} C_VEL
LIN {X 0,Y 193.189,Z 323.772,A -85,B 0,C 180,E1 -22015.847,E2 -22015.847} C_VEL
LIN {X 0,Y 194.953,Z 327.526,A -85,B 0,C 180,E1 -22016.475,E2 -22016.475} C_VEL
LIN {X 0,Y 201.726,Z 341.937,A -85,B 0,C 180,E1 -22018.334,E2 -22018.334} C_VEL
LIN {X 0,Y 206.688,Z 354.687,A -85,B 0,C 180,E1 -22019.683,E2 -22019.683} C_VEL
LIN {X 0,Y 208.586,Z 367.831,A -85,B 0,C 180,E1 -22020.499,E2 -22020.499} C_VEL
LIN {X 0,Y 208.016,Z 382.602,A -85,B 0,C 180,E1 -22020.983,E2 -22020.983} C_VEL
LIN {X 0,Y 207.159,Z 388.467,A -85,B 0,C 180,E1 -22021.069,E2 -22021.069} C_VEL
LIN {X 0,Y 204.192,Z 397.973,A -85,B 0,C 180,E1 -22021.001,E2 -22021.001} C_VEL
LIN {X 0,Y 201.021,Z 407.341,A -85,B 0,C 180,E1 -22021.1,E2 -22021.1} C_VEL
LIN {X 0,Y 199.843,Z 412.975,A -85,B 0,C 180,E1 -22021.454,E2 -22021.454} C_VEL
LIN {X 0,Y 198.305,Z 423.744,A -85,B 0,C 180,E1 -22022.567,E2 -22022.567} C_VEL
LIN {X 0,Y 196.775,Z 432.404,A -85,B 0,C 180,E1 -22023.77,E2 -22023.77} C_VEL
LIN {X 0,Y 194.95,Z 440.679,A -85,B 0,C 180,E1 -22025.224,E2 -22025.224} C_VEL
LIN {X 0,Y 192.98,Z 448.514,A -85,B 0,C 180,E1 -22026.953,E2 -22026.953} C_VEL
LIN {X 0,Y 190.92,Z 455.84,A -85,B 0,C 180,E1 -22028.967,E2 -22028.967} C_VEL
LIN {X 0,Y 188.71,Z 463.27,A -85,B 0,C 180,E1 -22031.545,E2 -22031.545} C_VEL
LIN {X 0,Y 186.877,Z 469.09,A -85,B 0,C 180,E1 -22034.178,E2 -22034.178} C_VEL
LIN {X 0,Y 185.468,Z 473.678,A -85,B 0,C 180,E1 -22036.859,E2 -22036.859} C_VEL
LIN {X 0,Y 184.569,Z 476.659,A -85,B 0,C 180,E1 -22039.025,E2 -22039.025} C_VEL
LIN {X 0,Y 183.916,Z 478.972,A -85,B 0,C 180,E1 -22041.208,E2 -22041.208} C_VEL
LIN {X 0,Y 183.457,Z 480.704,A -85,B 0,C 180,E1 -22043.401,E2 -22043.401} C_VEL
LIN {X 0,Y 183.129,Z 482.207,A -85,B 0,C 180,E1 -22046.204,E2 -22046.204} C_VEL
LIN {X 0,Y 183.035,Z 483,A -85,B 0,C 180,E1 -22050,E2 -22050} C_VEL
LIN {X 0,Y 183.101,Z 482.237,A -85,B 0,C 180,E1 -22053.661,E2 -22053.661} C_VEL
LIN {X 0,Y 183.409,Z 480.655,A -85,B 0,C 180,E1 -22056.601,E2 -22056.601} C_VEL
LIN {X 0,Y 184.206,Z 477.752,A -85,B 0,C 180,E1 -22059.886,E2 -22059.886} C_VEL
LIN {X 0,Y 185,Z 475.104,A -85,B 0,C 180,E1 -22062.06,E2 -22062.06} C_VEL
LIN {X 0,Y 186.543,Z 469.929,A -85,B 0,C 180,E1 -22065.291,E2 -22065.291} C_VEL
LIN {X 0,Y 188.707,Z 463.101,A -85,B 0,C 180,E1 -22068.455,E2 -22068.455} C_VEL
LIN {X 0,Y 190.931,Z 455.639,A -85,B 0,C 180,E1 -22071.031,E2 -22071.031} C_VEL
LIN {X 0,Y 192.961,Z 448.276,A -85,B 0,C 180,E1 -22073.05,E2 -22073.05} C_VEL
LIN {X 0,Y 194.965,Z 440.387,A -85,B 0,C 180,E1 -22074.774,E2 -22074.774} C_VEL
LIN {X 0,Y 196.702,Z 432.044,A -85,B 0,C 180,E1 -22076.24,E2 -22076.24} C_VEL
LIN {X 0,Y 198.595,Z 421.363,A -85,B 0,C 180,E1 -22077.676,E2 -22077.676} C_VEL
LIN {X 0,Y 200.037,Z 410.523,A -85,B 0,C 180,E1 -22078.67,E2 -22078.67} C_VEL
LIN {X 0,Y 200.941,Z 401.123,A -85,B 0,C 180,E1 -22079.245,E2 -22079.245} C_VEL
LIN {X 0,Y 202.167,Z 372.072,A -85,B 0,C 180,E1 -22080.296,E2 -22080.296} C_VEL
LIN {X 0,Y 202.132,Z 367.011,A -85,B 0,C 180,E1 -22080.506,E2 -22080.506} C_VEL
LIN {X 0,Y 200.487,Z 356.338,A -85,B 0,C 180,E1 -22081.22,E2 -22081.22} C_VEL
LIN {X 0,Y 194.391,Z 341.151,A -85,B 0,C 180,E1 -22082.967,E2 -22082.967} C_VEL
LIN {X 0,Y 187.702,Z 327.482,A -85,B 0,C 180,E1 -22084.923,E2 -22084.923} C_VEL
LIN {X 0,Y 185.887,Z 323.757,A -85,B 0,C 180,E1 -22085.618,E2 -22085.618} C_VEL
LIN {X 0,Y 185.556,Z 322.244,A -85,B 0,C 180,E1 -22086.728,E2 -22086.728} C_VEL
LIN {X 0,Y 185.458,Z 322.155,A -85,B 0,C 180,E1 -22090.72,E2 -22090.72} C_VEL
LIN {X 0,Y 185.453,Z 322.198,A -85,B 0,C 180,E1 -22096.056,E2 -22096.056} C_VEL
LIN {X 0,Y 185.451,Z 322.138,A -85,B 0,C 180,E1 -22099.891,E2 -22099.891} C_VEL
LIN {X 0,Y 185.497,Z 322.14,A -85,B 0,C 180,E1 -22102.714,E2 -22102.714} C_VEL
LIN {X 0,Y 185.527,Z 322.184,A -85,B 0,C 180,E1 -22107.972,E2 -22107.972} C_VEL
LIN {X 0,Y 185.543,Z 322.166,A -85,B 0,C 180,E1 -22110.595,E2 -22110.595} C_VEL
LIN {X 0,Y 185.559,Z 322.178,A -85,B 0,C 180,E1 -22115.379,E2 -22115.379} C_VEL
LIN {X 0,Y 185.621,Z 322.175,A -85,B 0,C 180,E1 -22121.179,E2 -22121.179} C_VEL
LIN {X 0,Y 185.692,Z 322.141,A -85,B 0,C 180,E1 -22126.875,E2 -22126.875} C_VEL
LIN {X 0,Y 185.97,Z 322.13,A -85,B 0,C 180,E1 -22131.306,E2 -22131.306} C_VEL
LIN {X 0,Y 186.168,Z 322.097,A -85,B 0,C 180,E1 -22137.837,E2 -22137.837} C_VEL
LIN {X 0,Y 186.373,Z 322.084,A -85,B 0,C 180,E1 -22140,E2 -22140} C_VEL
LIN {X 0,Y 185.868,Z 322.115,A -85,B 0,C 180,E1 -22144.337,E2 -22144.337} C_VEL
LIN {X 0,Y 185.964,Z 322.131,A -85,B 0,C 180,E1 -22148.695,E2 -22148.695} C_VEL
LIN {X 0,Y 185.693,Z 322.141,A -85,B 0,C 180,E1 -22153.126,E2 -22153.126} C_VEL
LIN {X 0,Y 185.621,Z 322.175,A -85,B 0,C 180,E1 -22158.821,E2 -22158.821} C_VEL
LIN {X 0,Y 185.558,Z 322.178,A -85,B 0,C 180,E1 -22164.635,E2 -22164.635} C_VEL
LIN {X 0,Y 185.541,Z 322.166,A -85,B 0,C 180,E1 -22169.5,E2 -22169.5} C_VEL
LIN {X 0,Y 185.494,Z 322.184,A -85,B 0,C 180,E1 -22174.634,E2 -22174.634} C_VEL
LIN {X 0,Y 185.497,Z 322.141,A -85,B 0,C 180,E1 -22177.315,E2 -22177.315} C_VEL
LIN {X 0,Y 185.458,Z 322.142,A -85,B 0,C 180,E1 -22180.721,E2 -22180.721} C_VEL
LIN {X 0,Y 185.453,Z 322.179,A -85,B 0,C 180,E1 -22186.058,E2 -22186.058} C_VEL
LIN {X 0,Y 185.454,Z 322.159,A -85,B 0,C 180,E1 -22189.893,E2 -22189.893} C_VEL
LIN {X 0,Y 185.576,Z 322.29,A -85,B 0,C 180,E1 -22193.454,E2 -22193.454} C_VEL
LIN {X 0,Y 185.97,Z 323.96,A -85,B 0,C 180,E1 -22194.498,E2 -22194.498} C_VEL
LIN {X 0,Y 189.72,Z 331.313,A -85,B 0,C 180,E1 -22195.719,E2 -22195.719} C_VEL
LIN {X 0,Y 196.965,Z 347.294,A -85,B 0,C 180,E1 -22197.822,E2 -22197.822} C_VEL
LIN {X 0,Y 200.719,Z 357.241,A -85,B 0,C 180,E1 -22198.902,E2 -22198.902} C_VEL
LIN {X 0,Y 202.271,Z 368.223,A -85,B 0,C 180,E1 -22199.611,E2 -22199.611} C_VEL
LIN {X 0,Y 200.939,Z 400.154,A -85,B 0,C 180,E1 -22200.746,E2 -22200.746} C_VEL
LIN {X 0,Y 200.069,Z 409.634,A -85,B 0,C 180,E1 -22201.303,E2 -22201.303} C_VEL
LIN {X 0,Y 198.889,Z 419.49,A -85,B 0,C 180,E1 -22202.184,E2 -22202.184} C_VEL
LIN {X 0,Y 197.128,Z 430.304,A -85,B 0,C 180,E1 -22203.536,E2 -22203.536} C_VEL
LIN {X 0,Y 195.002,Z 440.192,A -85,B 0,C 180,E1 -22205.231,E2 -22205.231} C_VEL
LIN {X 0,Y 193.006,Z 448.114,A -85,B 0,C 180,E1 -22206.956,E2 -22206.956} C_VEL
LIN {X 0,Y 191.461,Z 453.802,A -85,B 0,C 180,E1 -22208.465,E2 -22208.465} C_VEL
LIN {X 0,Y 189.558,Z 460.157,A -85,B 0,C 180,E1 -22210.508,E2 -22210.508} C_VEL
LIN {X 0,Y 187.963,Z 465.441,A -85,B 0,C 180,E1 -22212.596,E2 -22212.596} C_VEL
LIN {X 0,Y 186.588,Z 469.852,A -85,B 0,C 180,E1 -22214.713,E2 -22214.713} C_VEL
LIN {X 0,Y 185.031,Z 475.043,A -85,B 0,C 180,E1 -22217.942,E2 -22217.942} C_VEL
LIN {X 0,Y 184.215,Z 477.705,A -85,B 0,C 180,E1 -22220.115,E2 -22220.115} C_VEL
LIN {X 0,Y 183.411,Z 480.622,A -85,B 0,C 180,E1 -22223.399,E2 -22223.399} C_VEL
LIN {X 0,Y 183.102,Z 482.217,A -85,B 0,C 180,E1 -22226.339,E2 -22226.339} C_VEL
LIN {X 0,Y 183.035,Z 482.999,A -85,B 0,C 180,E1 -22230,E2 -22230} C_VEL
LIN {X 0,Y 183.097,Z 482.298,A -85,B 0,C 180,E1 -22233.634,E2 -22233.634} C_VEL
LIN {X 0,Y 183.411,Z 480.737,A -85,B 0,C 180,E1 -22236.601,E2 -22236.601} C_VEL
LIN {X 0,Y 184.206,Z 477.868,A -85,B 0,C 180,E1 -22239.886,E2 -22239.886} C_VEL
LIN {X 0,Y 184.994,Z 475.256,A -85,B 0,C 180,E1 -22242.06,E2 -22242.06} C_VEL
LIN {X 0,Y 186.544,Z 470.123,A -85,B 0,C 180,E1 -22245.291,E2 -22245.291} C_VEL
LIN {X 0,Y 188.335,Z 464.601,A -85,B 0,C 180,E1 -22247.93,E2 -22247.93} C_VEL
LIN {X 0,Y 190.392,Z 457.662,A -85,B 0,C 180,E1 -22250.528,E2 -22250.528} C_VEL
LIN {X 0,Y 192.673,Z 449.697,A -85,B 0,C 180,E1 -22252.802,E2 -22252.802} C_VEL
LIN {X 0,Y 194.648,Z 442.103,A -85,B 0,C 180,E1 -22254.533,E2 -22254.533} C_VEL
LIN {X 0,Y 196.477,Z 434.141,A -85,B 0,C 180,E1 -22255.987,E2 -22255.987} C_VEL
LIN {X 0,Y 198.047,Z 425.912,A -85,B 0,C 180,E1 -22257.186,E2 -22257.186} C_VEL
LIN {X 0,Y 199.315,Z 416.892,A -85,B 0,C 180,E1 -22258.217,E2 -22258.217} C_VEL
LIN {X 0,Y 200.39,Z 407.664,A -85,B 0,C 180,E1 -22258.975,E2 -22258.975} C_VEL
LIN {X 0,Y 201.144,Z 397.792,A -85,B 0,C 180,E1 -22259.512,E2 -22259.512} C_VEL
LIN {X 0,Y 202.319,Z 367.172,A -85,B 0,C 180,E1 -22260.583,E2 -22260.583} C_VEL
LIN {X 0,Y 200.58,Z 356.609,A -85,B 0,C 180,E1 -22261.31,E2 -22261.31} C_VEL
LIN {X 0,Y 194.737,Z 341.9,A -85,B 0,C 180,E1 -22262.991,E2 -22262.991} C_VEL
LIN {X 0,Y 188.708,Z 329.44,A -85,B 0,C 180,E1 -22264.75,E2 -22264.75} C_VEL
LIN {X 0,Y 186.004,Z 324.069,A -85,B 0,C 180,E1 -22265.649,E2 -22265.649} C_VEL
LIN {X 0,Y 185.582,Z 322.5,A -85,B 0,C 180,E1 -22266.528,E2 -22266.528} C_VEL
LIN {X 0,Y 185.498,Z 322.186,A -85,B 0,C 180,E1 -22267.314,E2 -22267.314} C_VEL
LIN {X 0,Y 185.459,Z 322.155,A -85,B 0,C 180,E1 -22270.72,E2 -22270.72} C_VEL
LIN {X 0,Y 185.453,Z 322.198,A -85,B 0,C 180,E1 -22276.056,E2 -22276.056} C_VEL
LIN {X 0,Y 185.448,Z 322.14,A -85,B 0,C 180,E1 -22279.89,E2 -22279.89} C_VEL
LIN {X 0,Y 185.498,Z 322.139,A -85,B 0,C 180,E1 -22282.713,E2 -22282.713} C_VEL
LIN {X 0,Y 185.527,Z 322.185,A -85,B 0,C 180,E1 -22287.972,E2 -22287.972} C_VEL
LIN {X 0,Y 185.544,Z 322.166,A -85,B 0,C 180,E1 -22290.595,E2 -22290.595} C_VEL
LIN {X 0,Y 185.559,Z 322.179,A -85,B 0,C 180,E1 -22295.378,E2 -22295.378} C_VEL
LIN {X 0,Y 185.621,Z 322.175,A -85,B 0,C 180,E1 -22301.179,E2 -22301.179} C_VEL
LIN {X 0,Y 185.693,Z 322.14,A -85,B 0,C 180,E1 -22306.874,E2 -22306.874} C_VEL
LIN {X 0,Y 185.97,Z 322.13,A -85,B 0,C 180,E1 -22311.305,E2 -22311.305} C_VEL
LIN {X 0,Y 186.168,Z 322.097,A -85,B 0,C 180,E1 -22317.836,E2 -22317.836} C_VEL
LIN {X 0,Y 186.373,Z 322.084,A -85,B 0,C 180,E1 -22320,E2 -22320} C_VEL
LIN {X 0,Y 185.868,Z 322.115,A -85,B 0,C 180,E1 -22324.337,E2 -22324.337} C_VEL
LIN {X 0,Y 185.964,Z 322.131,A -85,B 0,C 180,E1 -22328.694,E2 -22328.694} C_VEL
LIN {X 0,Y 185.692,Z 322.141,A -85,B 0,C 180,E1 -22333.125,E2 -22333.125} C_VEL
LIN {X 0,Y 185.621,Z 322.175,A -85,B 0,C 180,E1 -22338.821,E2 -22338.821} C_VEL
LIN {X 0,Y 185.557,Z 322.179,A -85,B 0,C 180,E1 -22344.635,E2 -22344.635} C_VEL
LIN {X 0,Y 185.54,Z 322.166,A -85,B 0,C 180,E1 -22349.5,E2 -22349.5} C_VEL
LIN {X 0,Y 185.493,Z 322.183,A -85,B 0,C 180,E1 -22354.633,E2 -22354.633} C_VEL
LIN {X 0,Y 185.496,Z 322.139,A -85,B 0,C 180,E1 -22357.315,E2 -22357.315} C_VEL
LIN {X 0,Y 185.457,Z 322.144,A -85,B 0,C 180,E1 -22360.721,E2 -22360.721} C_VEL
LIN {X 0,Y 185.451,Z 322.176,A -85,B 0,C 180,E1 -22366.057,E2 -22366.057} C_VEL
LIN {X 0,Y 185.452,Z 322.16,A -85,B 0,C 180,E1 -22369.892,E2 -22369.892} C_VEL
LIN {X 0,Y 185.575,Z 322.432,A -85,B 0,C 180,E1 -22373.466,E2 -22373.466} C_VEL
LIN {X 0,Y 185.951,Z 323.947,A -85,B 0,C 180,E1 -22374.358,E2 -22374.358} C_VEL
LIN {X 0,Y 189.578,Z 331.16,A -85,B 0,C 180,E1 -22375.555,E2 -22375.555} C_VEL
LIN {X 0,Y 196.002,Z 344.844,A -85,B 0,C 180,E1 -22377.419,E2 -22377.419} C_VEL
LIN {X 0,Y 200.875,Z 357.541,A -85,B 0,C 180,E1 -22378.825,E2 -22378.825} C_VEL
LIN {X 0,Y 202.399,Z 368.236,A -85,B 0,C 180,E1 -22379.518,E2 -22379.518} C_VEL
LIN {X 0,Y 201.012,Z 401.076,A -85,B 0,C 180,E1 -22380.694,E2 -22380.694} C_VEL
LIN {X 0,Y 199.866,Z 412.789,A -85,B 0,C 180,E1 -22381.437,E2 -22381.437} C_VEL
LIN {X 0,Y 199.843,Z 412.975,A -85,B 0,C 180,E1 -22381.454,E2 -22381.454} C_VEL
LIN {X 0,Y 199.032,Z 416.722,A -85,B 0,C 180,E1 -22381.75,E2 -22381.75} C_VEL
LIN {X 0,Y 196.203,Z 423.975,A -85,B 0,C 180,E1 -22382.275,E2 -22382.275} C_VEL
LIN {X 0,Y 190.226,Z 435.854,A -85,B 0,C 180,E1 -22383.469,E2 -22383.469} C_VEL
LIN {X 0,Y 188.54,Z 440.661,A -85,B 0,C 180,E1 -22384.316,E2 -22384.316} C_VEL
LIN {X 0,Y 186.481,Z 448.517,A -85,B 0,C 180,E1 -22386.101,E2 -22386.101} C_VEL
LIN {X 0,Y 184.318,Z 455.843,A -85,B 0,C 180,E1 -22388.176,E2 -22388.176} C_VEL
LIN {X 0,Y 181.978,Z 463.272,A -85,B 0,C 180,E1 -22390.837,E2 -22390.837} C_VEL
LIN {X 0,Y 180.059,Z 469.092,A -85,B 0,C 180,E1 -22393.562,E2 -22393.562} C_VEL
LIN {X 0,Y 178.538,Z 473.679,A -85,B 0,C 180,E1 -22396.339,E2 -22396.339} C_VEL
LIN {X 0,Y 177.588,Z 476.66,A -85,B 0,C 180,E1 -22398.588,E2 -22398.588} C_VEL
LIN {X 0,Y 176.888,Z 478.973,A -85,B 0,C 180,E1 -22400.856,E2 -22400.856} C_VEL
LIN {X 0,Y 176.409,Z 480.704,A -85,B 0,C 180,E1 -22403.136,E2 -22403.136} C_VEL
LIN {X 0,Y 175.995,Z 482.472,A -85,B 0,C 180,E1 -22406.681,E2 -22406.681} C_VEL
LIN {X 0,Y 175.95,Z 483,A -85,B 0,C 180,E1 -22410,E2 -22410} C_VEL
LIN {X 0,Y 175.97,Z 482.501,A -85,B 0,C 180,E1 -22413.176,E2 -22413.176} C_VEL
LIN {X 0,Y 176.353,Z 480.654,A -85,B 0,C 180,E1 -22416.866,E2 -22416.866} C_VEL
LIN {X 0,Y 177.208,Z 477.751,A -85,B 0,C 180,E1 -22420.28,E2 -22420.28} C_VEL
LIN {X 0,Y 178.045,Z 475.103,A -85,B 0,C 180,E1 -22422.539,E2 -22422.539} C_VEL
LIN {X 0,Y 179.702,Z 469.928,A -85,B 0,C 180,E1 -22425.888,E2 -22425.888} C_VEL
LIN {X 0,Y 181.976,Z 463.099,A -85,B 0,C 180,E1 -22429.164,E2 -22429.164} C_VEL
LIN {X 0,Y 184.329,Z 455.636,A -85,B 0,C 180,E1 -22431.823,E2 -22431.823} C_VEL
LIN {X 0,Y 186.453,Z 448.273,A -85,B 0,C 180,E1 -22433.903,E2 -22433.903} C_VEL
LIN {X 0,Y 188.544,Z 440.383,A -85,B 0,C 180,E1 -22435.678,E2 -22435.678} C_VEL
LIN {X 0,Y 190.687,Z 430.584,A -85,B 0,C 180,E1 -22437.423,E2 -22437.423} C_VEL
LIN {X 0,Y 192.667,Z 419.021,A -85,B 0,C 180,E1 -22438.901,E2 -22438.901} C_VEL
LIN {X 0,Y 193.93,Z 409.68,A -85,B 0,C 180,E1 -22439.736,E2 -22439.736} C_VEL
LIN {X 0,Y 194.83,Z 399.808,A -85,B 0,C 180,E1 -22440.332,E2 -22440.332} C_VEL
LIN {X 0,Y 196.093,Z 368.435,A -85,B 0,C 180,E1 -22441.49,E2 -22441.49} C_VEL
LIN {X 0,Y 194.643,Z 358.896,A -85,B 0,C 180,E1 -22442.158,E2 -22442.158} C_VEL
LIN {X 0,Y 189.144,Z 344.998,A -85,B 0,C 180,E1 -22443.831,E2 -22443.831} C_VEL
LIN {X 0,Y 182.771,Z 331.736,A -85,B 0,C 180,E1 -22445.806,E2 -22445.806} C_VEL
LIN {X 0,Y 178.713,Z 324.173,A -85,B 0,C 180,E1 -22447.185,E2 -22447.185} C_VEL
LIN {X 0,Y 178.451,Z 323.255,A -85,B 0,C 180,E1 -22447.643,E2 -22447.643} C_VEL
LIN {X 0,Y 178.39,Z 323.034,A -85,B 0,C 180,E1 -22452.046,E2 -22452.046} C_VEL
LIN {X 0,Y 178.388,Z 323.076,A -85,B 0,C 180,E1 -22455.164,E2 -22455.164} C_VEL
LIN {X 0,Y 178.393,Z 323.031,A -85,B 0,C 180,E1 -22458.461,E2 -22458.461} C_VEL
LIN {X 0,Y 178.415,Z 323.036,A -85,B 0,C 180,E1 -22463.782,E2 -22463.782} C_VEL
LIN {X 0,Y 178.48,Z 323.066,A -85,B 0,C 180,E1 -22466.546,E2 -22466.546} C_VEL
LIN {X 0,Y 178.436,Z 323.058,A -85,B 0,C 180,E1 -22471.794,E2 -22471.794} C_VEL
LIN {X 0,Y 178.501,Z 323.059,A -85,B 0,C 180,E1 -22474.896,E2 -22474.896} C_VEL
LIN {X 0,Y 178.601,Z 323.049,A -85,B 0,C 180,E1 -22481.651,E2 -22481.651} C_VEL
LIN {X 0,Y 178.62,Z 323.019,A -85,B 0,C 180,E1 -22486.345,E2 -22486.345} C_VEL
LIN {X 0,Y 178.9,Z 323.011,A -85,B 0,C 180,E1 -22490.959,E2 -22490.959} C_VEL
LIN {X 0,Y 179.116,Z 322.975,A -85,B 0,C 180,E1 -22497.752,E2 -22497.752} C_VEL
LIN {X 0,Y 179.338,Z 322.96,A -85,B 0,C 180,E1 -22500,E2 -22500} C_VEL
LIN {X 0,Y 178.817,Z 322.992,A -85,B 0,C 180,E1 -22504.509,E2 -22504.509} C_VEL
LIN {X 0,Y 178.896,Z 323.012,A -85,B 0,C 180,E1 -22509.041,E2 -22509.041} C_VEL
LIN {X 0,Y 178.62,Z 323.019,A -85,B 0,C 180,E1 -22513.655,E2 -22513.655} C_VEL
LIN {X 0,Y 178.55,Z 323.054,A -85,B 0,C 180,E1 -22519.151,E2 -22519.151} C_VEL
LIN {X 0,Y 178.502,Z 323.059,A -85,B 0,C 180,E1 -22525.104,E2 -22525.104} C_VEL
LIN {X 0,Y 178.457,Z 323.051,A -85,B 0,C 180,E1 -22530.795,E2 -22530.795} C_VEL
LIN {X 0,Y 178.48,Z 323.062,A -85,B 0,C 180,E1 -22534.219,E2 -22534.219} C_VEL
LIN {X 0,Y 178.384,Z 323.012,A -85,B 0,C 180,E1 -22539.078,E2 -22539.078} C_VEL
LIN {X 0,Y 178.391,Z 323.04,A -85,B 0,C 180,E1 -22542.048,E2 -22542.048} C_VEL
LIN {X 0,Y 178.389,Z 323.072,A -85,B 0,C 180,E1 -22545.166,E2 -22545.166} C_VEL
LIN {X 0,Y 178.395,Z 323.032,A -85,B 0,C 180,E1 -22548.463,E2 -22548.463} C_VEL
LIN {X 0,Y 178.498,Z 323.334,A -85,B 0,C 180,E1 -22552.493,E2 -22552.493} C_VEL
LIN {X 0,Y 178.765,Z 324.32,A -85,B 0,C 180,E1 -22552.894,E2 -22552.894} C_VEL
LIN {X 0,Y 184.871,Z 335.73,A -85,B 0,C 180,E1 -22554.893,E2 -22554.893} C_VEL
LIN {X 0,Y 191.802,Z 351.443,A -85,B 0,C 180,E1 -22557.027,E2 -22557.027} C_VEL
LIN {X 0,Y 194.968,Z 360.11,A -85,B 0,C 180,E1 -22557.998,E2 -22557.998} C_VEL
LIN {X 0,Y 196.172,Z 368.919,A -85,B 0,C 180,E1 -22558.589,E2 -22558.589} C_VEL
LIN {X 0,Y 194.781,Z 400.276,A -85,B 0,C 180,E1 -22559.732,E2 -22559.732} C_VEL
LIN {X 0,Y 193.815,Z 410.457,A -85,B 0,C 180,E1 -22560.359,E2 -22560.359} C_VEL
LIN {X 0,Y 192.366,Z 421.41,A -85,B 0,C 180,E1 -22561.4,E2 -22561.4} C_VEL
LIN {X 0,Y 190.472,Z 431.812,A -85,B 0,C 180,E1 -22562.832,E2 -22562.832} C_VEL
LIN {X 0,Y 188.58,Z 440.196,A -85,B 0,C 180,E1 -22564.327,E2 -22564.327} C_VEL
LIN {X 0,Y 186.507,Z 448.117,A -85,B 0,C 180,E1 -22566.104,E2 -22566.104} C_VEL
LIN {X 0,Y 184.88,Z 453.805,A -85,B 0,C 180,E1 -22567.658,E2 -22567.658} C_VEL
LIN {X 0,Y 182.888,Z 460.16,A -85,B 0,C 180,E1 -22569.767,E2 -22569.767} C_VEL
LIN {X 0,Y 181.189,Z 465.443,A -85,B 0,C 180,E1 -22571.923,E2 -22571.923} C_VEL
LIN {X 0,Y 179.745,Z 469.854,A -85,B 0,C 180,E1 -22574.116,E2 -22574.116} C_VEL
LIN {X 0,Y 178.075,Z 475.044,A -85,B 0,C 180,E1 -22577.464,E2 -22577.464} C_VEL
LIN {X 0,Y 177.219,Z 477.706,A -85,B 0,C 180,E1 -22579.72,E2 -22579.72} C_VEL
LIN {X 0,Y 176.355,Z 480.623,A -85,B 0,C 180,E1 -22583.134,E2 -22583.134} C_VEL
LIN {X 0,Y 175.971,Z 482.483,A -85,B 0,C 180,E1 -22586.824,E2 -22586.824} C_VEL
LIN {X 0,Y 175.95,Z 482.999,A -85,B 0,C 180,E1 -22590,E2 -22590} C_VEL
LIN {X 0,Y 175.996,Z 482.49,A -85,B 0,C 180,E1 -22593.319,E2 -22593.319} C_VEL
LIN {X 0,Y 176.355,Z 480.736,A -85,B 0,C 180,E1 -22596.866,E2 -22596.866} C_VEL
LIN {X 0,Y 177.208,Z 477.867,A -85,B 0,C 180,E1 -22600.28,E2 -22600.28} C_VEL
LIN {X 0,Y 178.036,Z 475.255,A -85,B 0,C 180,E1 -22602.539,E2 -22602.539} C_VEL
LIN {X 0,Y 179.707,Z 470.121,A -85,B 0,C 180,E1 -22605.888,E2 -22605.888} C_VEL
LIN {X 0,Y 181.562,Z 464.599,A -85,B 0,C 180,E1 -22608.623,E2 -22608.623} C_VEL
LIN {X 0,Y 183.768,Z 457.659,A -85,B 0,C 180,E1 -22611.304,E2 -22611.304} C_VEL
LIN {X 0,Y 186.164,Z 449.693,A -85,B 0,C 180,E1 -22613.647,E2 -22613.647} C_VEL
LIN {X 0,Y 188.218,Z 442.099,A -85,B 0,C 180,E1 -22615.429,E2 -22615.429} C_VEL
LIN {X 0,Y 190.125,Z 434.136,A -85,B 0,C 180,E1 -22616.924,E2 -22616.924} C_VEL
LIN {X 0,Y 191.764,Z 425.905,A -85,B 0,C 180,E1 -22618.154,E2 -22618.154} C_VEL
LIN {X 0,Y 193.075,Z 417.116,A -85,B 0,C 180,E1 -22619.187,E2 -22619.187} C_VEL
LIN {X 0,Y 194.173,Z 408.082,A -85,B 0,C 180,E1 -22619.958,E2 -22619.958} C_VEL
LIN {X 0,Y 194.955,Z 398.493,A -85,B 0,C 180,E1 -22620.505,E2 -22620.505} C_VEL
LIN {X 0,Y 196.188,Z 368.22,A -85,B 0,C 180,E1 -22621.602,E2 -22621.602} C_VEL
LIN {X 0,Y 194.707,Z 358.93,A -85,B 0,C 180,E1 -22622.267,E2 -22622.267} C_VEL
LIN {X 0,Y 189.124,Z 344.937,A -85,B 0,C 180,E1 -22623.965,E2 -22623.965} C_VEL
LIN {X 0,Y 183.646,Z 333.457,A -85,B 0,C 180,E1 -22625.662,E2 -22625.662} C_VEL
LIN {X 0,Y 179.66,Z 326.217,A -85,B 0,C 180,E1 -22626.933,E2 -22626.933} C_VEL
LIN {X 0,Y 178.587,Z 323.79,A -85,B 0,C 180,E1 -22627.449,E2 -22627.449} C_VEL
LIN {X 0,Y 178.429,Z 323.144,A -85,B 0,C 180,E1 -22628.022,E2 -22628.022} C_VEL
LIN {X 0,Y 178.391,Z 323.033,A -85,B 0,C 180,E1 -22632.046,E2 -22632.046} C_VEL
LIN {X 0,Y 178.389,Z 323.075,A -85,B 0,C 180,E1 -22635.164,E2 -22635.164} C_VEL
LIN {X 0,Y 178.393,Z 323.033,A -85,B 0,C 180,E1 -22638.461,E2 -22638.461} C_VEL
LIN {X 0,Y 178.416,Z 323.034,A -85,B 0,C 180,E1 -22643.781,E2 -22643.781} C_VEL
LIN {X 0,Y 178.481,Z 323.065,A -85,B 0,C 180,E1 -22646.545,E2 -22646.545} C_VEL
LIN {X 0,Y 178.437,Z 323.057,A -85,B 0,C 180,E1 -22651.794,E2 -22651.794} C_VEL
LIN {X 0,Y 178.502,Z 323.06,A -85,B 0,C 180,E1 -22654.896,E2 -22654.896} C_VEL
LIN {X 0,Y 178.601,Z 323.049,A -85,B 0,C 180,E1 -22661.651,E2 -22661.651} C_VEL
LIN {X 0,Y 178.62,Z 323.019,A -85,B 0,C 180,E1 -22666.345,E2 -22666.345} C_VEL
LIN {X 0,Y 178.901,Z 323.011,A -85,B 0,C 180,E1 -22670.959,E2 -22670.959} C_VEL
LIN {X 0,Y 179.116,Z 322.975,A -85,B 0,C 180,E1 -22677.751,E2 -22677.751} C_VEL
LIN {X 0,Y 179.338,Z 322.96,A -85,B 0,C 180,E1 -22680,E2 -22680} C_VEL
LIN {X 0,Y 178.817,Z 322.992,A -85,B 0,C 180,E1 -22684.508,E2 -22684.508} C_VEL
LIN {X 0,Y 178.896,Z 323.012,A -85,B 0,C 180,E1 -22689.041,E2 -22689.041} C_VEL
LIN {X 0,Y 178.619,Z 323.019,A -85,B 0,C 180,E1 -22693.655,E2 -22693.655} C_VEL
LIN {X 0,Y 178.549,Z 323.053,A -85,B 0,C 180,E1 -22699.151,E2 -22699.151} C_VEL
LIN {X 0,Y 178.501,Z 323.06,A -85,B 0,C 180,E1 -22705.104,E2 -22705.104} C_VEL
LIN {X 0,Y 178.456,Z 323.052,A -85,B 0,C 180,E1 -22710.795,E2 -22710.795} C_VEL
LIN {X 0,Y 178.479,Z 323.061,A -85,B 0,C 180,E1 -22714.218,E2 -22714.218} C_VEL
LIN {X 0,Y 178.383,Z 323.012,A -85,B 0,C 180,E1 -22719.078,E2 -22719.078} C_VEL
LIN {X 0,Y 178.39,Z 323.043,A -85,B 0,C 180,E1 -22722.047,E2 -22722.047} C_VEL
LIN {X 0,Y 178.388,Z 323.07,A -85,B 0,C 180,E1 -22725.166,E2 -22725.166} C_VEL
LIN {X 0,Y 178.394,Z 323.032,A -85,B 0,C 180,E1 -22728.462,E2 -22728.462} C_VEL
LIN {X 0,Y 178.478,Z 323.365,A -85,B 0,C 180,E1 -22732.365,E2 -22732.365} C_VEL
LIN {X 0,Y 178.693,Z 324.192,A -85,B 0,C 180,E1 -22732.717,E2 -22732.717} C_VEL
LIN {X 0,Y 184.26,Z 334.703,A -85,B 0,C 180,E1 -22734.578,E2 -22734.578} C_VEL
LIN {X 0,Y 189.874,Z 346.659,A -85,B 0,C 180,E1 -22736.309,E2 -22736.309} C_VEL
LIN {X 0,Y 195.012,Z 359.906,A -85,B 0,C 180,E1 -22737.877,E2 -22737.877} C_VEL
LIN {X 0,Y 196.246,Z 368.609,A -85,B 0,C 180,E1 -22738.47,E2 -22738.47} C_VEL
LIN {X 0,Y 194.846,Z 401.091,A -85,B 0,C 180,E1 -22739.671,E2 -22739.671} C_VEL
LIN {X 0,Y 193.643,Z 413.021,A -85,B 0,C 180,E1 -22740.454,E2 -22740.454} C_VEL
LIN {X 0,Y 192.034,Z 423.75,A -85,B 0,C 180,E1 -22741.591,E2 -22741.591} C_VEL
LIN {X 0,Y 190.442,Z 432.408,A -85,B 0,C 180,E1 -22742.827,E2 -22742.827} C_VEL
LIN {X 0,Y 188.54,Z 440.661,A -85,B 0,C 180,E1 -22744.316,E2 -22744.316} C_VEL
LIN {X 0,Y 186.786,Z 445.517,A -85,B 0,C 180,E1 -22745.273,E2 -22745.273} C_VEL
LIN {X 0,Y 182.071,Z 452.752,A -85,B 0,C 180,E1 -22746.805,E2 -22746.805} C_VEL
LIN {X 0,Y 177.265,Z 459.332,A -85,B 0,C 180,E1 -22748.601,E2 -22748.601} C_VEL
LIN {X 0,Y 175.393,Z 462.945,A -85,B 0,C 180,E1 -22749.945,E2 -22749.945} C_VEL
LIN {X 0,Y 173.27,Z 469.093,A -85,B 0,C 180,E1 -22752.899,E2 -22752.899} C_VEL
LIN {X 0,Y 171.637,Z 473.68,A -85,B 0,C 180,E1 -22755.778,E2 -22755.778} C_VEL
LIN {X 0,Y 170.629,Z 476.661,A -85,B 0,C 180,E1 -22758.116,E2 -22758.116} C_VEL
LIN {X 0,Y 169.884,Z 478.974,A -85,B 0,C 180,E1 -22760.475,E2 -22760.475} C_VEL
LIN {X 0,Y 169.36,Z 480.705,A -85,B 0,C 180,E1 -22762.849,E2 -22762.849} C_VEL
LIN {X 0,Y 168.891,Z 482.632,A -85,B 0,C 180,E1 -22767.079,E2 -22767.079} C_VEL
LIN {X 0,Y 168.85,Z 483,A -85,B 0,C 180,E1 -22770,E2 -22770} C_VEL
LIN {X 0,Y 168.891,Z 482.615,A -85,B 0,C 180,E1 -22772.921,E2 -22772.921} C_VEL
LIN {X 0,Y 169.296,Z 480.654,A -85,B 0,C 180,E1 -22777.154,E2 -22777.154} C_VEL
LIN {X 0,Y 170.23,Z 477.75,A -85,B 0,C 180,E1 -22780.707,E2 -22780.707} C_VEL
LIN {X 0,Y 171.113,Z 475.102,A -85,B 0,C 180,E1 -22783.055,E2 -22783.055} C_VEL
LIN {X 0,Y 172.89,Z 469.926,A -85,B 0,C 180,E1 -22786.532,E2 -22786.532} C_VEL
LIN {X 0,Y 175.285,Z 463.097,A -85,B 0,C 180,E1 -22789.925,E2 -22789.925} C_VEL
LIN {X 0,Y 177.767,Z 455.633,A -85,B 0,C 180,E1 -22792.672,E2 -22792.672} C_VEL
LIN {X 0,Y 179.991,Z 448.27,A -85,B 0,C 180,E1 -22794.818,E2 -22794.818} C_VEL
LIN {X 0,Y 182.169,Z 440.38,A -85,B 0,C 180,E1 -22796.646,E2 -22796.646} C_VEL
LIN {X 0,Y 184.332,Z 431.006,A -85,B 0,C 180,E1 -22798.364,E2 -22798.364} C_VEL
LIN {X 0,Y 186.24,Z 420.689,A -85,B 0,C 180,E1 -22799.781,E2 -22799.781} C_VEL
LIN {X 0,Y 187.814,Z 409.67,A -85,B 0,C 180,E1 -22800.808,E2 -22800.808} C_VEL
LIN {X 0,Y 188.737,Z 399.792,A -85,B 0,C 180,E1 -22801.42,E2 -22801.42} C_VEL
LIN {X 0,Y 190.033,Z 369.288,A -85,B 0,C 180,E1 -22802.578,E2 -22802.578} C_VEL
LIN {X 0,Y 188.875,Z 361.449,A -85,B 0,C 180,E1 -22803.151,E2 -22803.151} C_VEL
LIN {X 0,Y 183.565,Z 347.987,A -85,B 0,C 180,E1 -22804.865,E2 -22804.865} C_VEL
LIN {X 0,Y 177.478,Z 335.22,A -85,B 0,C 180,E1 -22806.875,E2 -22806.875} C_VEL
LIN {X 0,Y 173.443,Z 328.147,A -85,B 0,C 180,E1 -22808.245,E2 -22808.245} C_VEL
LIN {X 0,Y 171.987,Z 326.097,A -85,B 0,C 180,E1 -22808.739,E2 -22808.739} C_VEL
LIN {X 0,Y 171.437,Z 324.495,A -85,B 0,C 180,E1 -22809.148,E2 -22809.148} C_VEL
LIN {X 0,Y 171.334,Z 323.965,A -85,B 0,C 180,E1 -22809.808,E2 -22809.808} C_VEL
LIN {X 0,Y 171.315,Z 323.938,A -85,B 0,C 180,E1 -22814.218,E2 -22814.218} C_VEL
LIN {X 0,Y 171.326,Z 323.901,A -85,B 0,C 180,E1 -22818.979,E2 -22818.979} C_VEL
LIN {X 0,Y 171.355,Z 323.889,A -85,B 0,C 180,E1 -22822.033,E2 -22822.033} C_VEL
LIN {X 0,Y 171.394,Z 323.934,A -85,B 0,C 180,E1 -22825.093,E2 -22825.093} C_VEL
LIN {X 0,Y 171.404,Z 323.925,A -85,B 0,C 180,E1 -22830.526,E2 -22830.526} C_VEL
LIN {X 0,Y 171.422,Z 323.931,A -85,B 0,C 180,E1 -22835.797,E2 -22835.797} C_VEL
LIN {X 0,Y 171.503,Z 323.931,A -85,B 0,C 180,E1 -22840.863,E2 -22840.863} C_VEL
LIN {X 0,Y 171.535,Z 323.901,A -85,B 0,C 180,E1 -22845.77,E2 -22845.77} C_VEL
LIN {X 0,Y 171.839,Z 323.892,A -85,B 0,C 180,E1 -22850.585,E2 -22850.585} C_VEL
LIN {X 0,Y 171.773,Z 323.868,A -85,B 0,C 180,E1 -22855.307,E2 -22855.307} C_VEL
LIN {X 0,Y 172.303,Z 323.836,A -85,B 0,C 180,E1 -22860,E2 -22860} C_VEL
LIN {X 0,Y 171.848,Z 323.875,A -85,B 0,C 180,E1 -22867.048,E2 -22867.048} C_VEL
LIN {X 0,Y 171.762,Z 323.894,A -85,B 0,C 180,E1 -22870.892,E2 -22870.892} C_VEL
LIN {X 0,Y 171.499,Z 323.927,A -85,B 0,C 180,E1 -22876.67,E2 -22876.67} C_VEL
LIN {X 0,Y 171.475,Z 323.932,A -85,B 0,C 180,E1 -22879.499,E2 -22879.499} C_VEL
LIN {X 0,Y 171.432,Z 323.942,A -85,B 0,C 180,E1 -22885.593,E2 -22885.593} C_VEL
LIN {X 0,Y 171.414,Z 323.926,A -85,B 0,C 180,E1 -22890.573,E2 -22890.573} C_VEL
LIN {X 0,Y 171.389,Z 323.933,A -85,B 0,C 180,E1 -22895.036,E2 -22895.036} C_VEL
LIN {X 0,Y 171.34,Z 323.887,A -85,B 0,C 180,E1 -22898.801,E2 -22898.801} C_VEL
LIN {X 0,Y 171.316,Z 323.959,A -85,B 0,C 180,E1 -22904.219,E2 -22904.219} C_VEL
LIN {X 0,Y 171.328,Z 323.91,A -85,B 0,C 180,E1 -22908.98,E2 -22908.98} C_VEL
LIN {X 0,Y 171.383,Z 324.251,A -85,B 0,C 180,E1 -22910.748,E2 -22910.748} C_VEL
LIN {X 0,Y 171.582,Z 325.072,A -85,B 0,C 180,E1 -22911.1,E2 -22911.1} C_VEL
LIN {X 0,Y 173.25,Z 327.964,A -85,B 0,C 180,E1 -22911.74,E2 -22911.74} C_VEL
LIN {X 0,Y 174.546,Z 329.903,A -85,B 0,C 180,E1 -22912.174,E2 -22912.174} C_VEL
LIN {X 0,Y 179.75,Z 339.655,A -85,B 0,C 180,E1 -22913.926,E2 -22913.926} C_VEL
LIN {X 0,Y 186.164,Z 354.296,A -85,B 0,C 180,E1 -22916.023,E2 -22916.023} C_VEL
LIN {X 0,Y 189.127,Z 362.175,A -85,B 0,C 180,E1 -22916.977,E2 -22916.977} C_VEL
LIN {X 0,Y 190.083,Z 370.787,A -85,B 0,C 180,E1 -22917.542,E2 -22917.542} C_VEL
LIN {X 0,Y 188.698,Z 400.343,A -85,B 0,C 180,E1 -22918.651,E2 -22918.651} C_VEL
LIN {X 0,Y 187.636,Z 410.855,A -85,B 0,C 180,E1 -22919.316,E2 -22919.316} C_VEL
LIN {X 0,Y 185.883,Z 423.013,A -85,B 0,C 180,E1 -22920.561,E2 -22920.561} C_VEL
LIN {X 0,Y 184.194,Z 431.817,A -85,B 0,C 180,E1 -22921.825,E2 -22921.825} C_VEL
LIN {X 0,Y 182.199,Z 440.201,A -85,B 0,C 180,E1 -22923.359,E2 -22923.359} C_VEL
LIN {X 0,Y 180.048,Z 448.121,A -85,B 0,C 180,E1 -22925.19,E2 -22925.19} C_VEL
LIN {X 0,Y 177.803,Z 455.509,A -85,B 0,C 180,E1 -22927.333,E2 -22927.333} C_VEL
LIN {X 0,Y 175.314,Z 462.995,A -85,B 0,C 180,E1 -22930.078,E2 -22930.078} C_VEL
LIN {X 0,Y 172.929,Z 469.855,A -85,B 0,C 180,E1 -22933.472,E2 -22933.472} C_VEL
LIN {X 0,Y 171.144,Z 475.046,A -85,B 0,C 180,E1 -22936.947,E2 -22936.947} C_VEL
LIN {X 0,Y 170.245,Z 477.707,A -85,B 0,C 180,E1 -22939.294,E2 -22939.294} C_VEL
LIN {X 0,Y 169.298,Z 480.623,A -85,B 0,C 180,E1 -22942.846,E2 -22942.846} C_VEL
LIN {X 0,Y 168.892,Z 482.605,A -85,B 0,C 180,E1 -22947.079,E2 -22947.079} C_VEL
LIN {X 0,Y 168.85,Z 482.999,A -85,B 0,C 180,E1 -22950,E2 -22950} C_VEL
LIN {X 0,Y 168.892,Z 482.641,A -85,B 0,C 180,E1 -22952.921,E2 -22952.921} C_VEL
LIN {X 0,Y 169.298,Z 480.735,A -85,B 0,C 180,E1 -22957.154,E2 -22957.154} C_VEL
LIN {X 0,Y 170.231,Z 477.866,A -85,B 0,C 180,E1 -22960.707,E2 -22960.707} C_VEL
LIN {X 0,Y 171.102,Z 475.253,A -85,B 0,C 180,E1 -22963.056,E2 -22963.056} C_VEL
LIN {X 0,Y 172.896,Z 470.12,A -85,B 0,C 180,E1 -22966.531,E2 -22966.531} C_VEL
LIN {X 0,Y 174.832,Z 464.598,A -85,B 0,C 180,E1 -22969.368,E2 -22969.368} C_VEL
LIN {X 0,Y 177.182,Z 457.657,A -85,B 0,C 180,E1 -22972.136,E2 -22972.136} C_VEL
LIN {X 0,Y 179.694,Z 449.69,A -85,B 0,C 180,E1 -22974.554,E2 -22974.554} C_VEL
LIN {X 0,Y 181.839,Z 442.095,A -85,B 0,C 180,E1 -22976.389,E2 -22976.389} C_VEL
LIN {X 0,Y 183.813,Z 434.131,A -85,B 0,C 180,E1 -22977.928,E2 -22977.928} C_VEL
LIN {X 0,Y 185.442,Z 426.439,A -85,B 0,C 180,E1 -22979.115,E2 -22979.115} C_VEL
LIN {X 0,Y 186.899,Z 417.291,A -85,B 0,C 180,E1 -22980.227,E2 -22980.227} C_VEL
LIN {X 0,Y 187.965,Z 409.069,A -85,B 0,C 180,E1 -22980.961,E2 -22980.961} C_VEL
LIN {X 0,Y 188.8,Z 399.611,A -85,B 0,C 180,E1 -22981.543,E2 -22981.543} C_VEL
LIN {X 0,Y 190.169,Z 369.369,A -85,B 0,C 180,E1 -22982.673,E2 -22982.673} C_VEL
LIN {X 0,Y 188.896,Z 361.354,A -85,B 0,C 180,E1 -22983.277,E2 -22983.277} C_VEL
LIN {X 0,Y 183.526,Z 347.816,A -85,B 0,C 180,E1 -22985.015,E2 -22985.015} C_VEL
LIN {X 0,Y 178.142,Z 336.42,A -85,B 0,C 180,E1 -22986.796,E2 -22986.796} C_VEL
LIN {X 0,Y 173.641,Z 328.377,A -85,B 0,C 180,E1 -22988.328,E2 -22988.328} C_VEL
LIN {X 0,Y 171.781,Z 325.662,A -85,B 0,C 180,E1 -22988.982,E2 -22988.982} C_VEL
LIN {X 0,Y 171.377,Z 324.279,A -85,B 0,C 180,E1 -22989.428,E2 -22989.428} C_VEL
LIN {X 0,Y 171.328,Z 323.911,A -85,B 0,C 180,E1 -22991.02,E2 -22991.02} C_VEL
LIN {X 0,Y 171.316,Z 323.959,A -85,B 0,C 180,E1 -22995.781,E2 -22995.781} C_VEL
LIN {X 0,Y 171.338,Z 323.887,A -85,B 0,C 180,E1 -23001.199,E2 -23001.199} C_VEL
LIN {X 0,Y 171.395,Z 323.931,A -85,B 0,C 180,E1 -23005.092,E2 -23005.092} C_VEL
LIN {X 0,Y 171.405,Z 323.925,A -85,B 0,C 180,E1 -23010.526,E2 -23010.526} C_VEL
LIN {X 0,Y 171.423,Z 323.932,A -85,B 0,C 180,E1 -23015.796,E2 -23015.796} C_VEL
LIN {X 0,Y 171.503,Z 323.93,A -85,B 0,C 180,E1 -23020.863,E2 -23020.863} C_VEL
LIN {X 0,Y 171.536,Z 323.901,A -85,B 0,C 180,E1 -23025.769,E2 -23025.769} C_VEL
LIN {X 0,Y 171.839,Z 323.892,A -85,B 0,C 180,E1 -23030.584,E2 -23030.584} C_VEL
LIN {X 0,Y 171.773,Z 323.868,A -85,B 0,C 180,E1 -23035.306,E2 -23035.306} C_VEL
LIN {X 0,Y 172.303,Z 323.836,A -85,B 0,C 180,E1 -23040,E2 -23040} C_VEL
LIN {X 0,Y 171.847,Z 323.875,A -85,B 0,C 180,E1 -23047.047,E2 -23047.047} C_VEL
LIN {X 0,Y 171.762,Z 323.894,A -85,B 0,C 180,E1 -23050.891,E2 -23050.891} C_VEL
LIN {X 0,Y 171.499,Z 323.928,A -85,B 0,C 180,E1 -23056.67,E2 -23056.67} C_VEL
LIN {X 0,Y 171.474,Z 323.931,A -85,B 0,C 180,E1 -23059.498,E2 -23059.498} C_VEL
LIN {X 0,Y 171.431,Z 323.943,A -85,B 0,C 180,E1 -23065.592,E2 -23065.592} C_VEL
LIN {X 0,Y 171.413,Z 323.927,A -85,B 0,C 180,E1 -23070.573,E2 -23070.573} C_VEL
LIN {X 0,Y 171.388,Z 323.93,A -85,B 0,C 180,E1 -23075.035,E2 -23075.035} C_VEL
LIN {X 0,Y 171.339,Z 323.887,A -85,B 0,C 180,E1 -23078.801,E2 -23078.801} C_VEL
LIN {X 0,Y 171.315,Z 323.959,A -85,B 0,C 180,E1 -23084.219,E2 -23084.219} C_VEL
LIN {X 0,Y 171.326,Z 323.911,A -85,B 0,C 180,E1 -23088.98,E2 -23088.98} C_VEL
LIN {X 0,Y 171.37,Z 324.223,A -85,B 0,C 180,E1 -23090.574,E2 -23090.574} C_VEL
LIN {X 0,Y 171.733,Z 325.481,A -85,B 0,C 180,E1 -23091.037,E2 -23091.037} C_VEL
LIN {X 0,Y 173.447,Z 328.183,A -85,B 0,C 180,E1 -23091.656,E2 -23091.656} C_VEL
LIN {X 0,Y 177.174,Z 334.73,A -85,B 0,C 180,E1 -23092.931,E2 -23092.931} C_VEL
LIN {X 0,Y 182.389,Z 345.316,A -85,B 0,C 180,E1 -23094.662,E2 -23094.662} C_VEL
LIN {X 0,Y 187.413,Z 357.35,A -85,B 0,C 180,E1 -23096.289,E2 -23096.289} C_VEL
LIN {X 0,Y 189.281,Z 362.773,A -85,B 0,C 180,E1 -23096.907,E2 -23096.907} C_VEL
LIN {X 0,Y 190.226,Z 370.266,A -85,B 0,C 180,E1 -23097.422,E2 -23097.422} C_VEL
LIN {X 0,Y 188.816,Z 399.938,A -85,B 0,C 180,E1 -23098.524,E2 -23098.524} C_VEL
LIN {X 0,Y 187.924,Z 409.504,A -85,B 0,C 180,E1 -23099.118,E2 -23099.118} C_VEL
LIN {X 0,Y 186.538,Z 419.66,A -85,B 0,C 180,E1 -23100.059,E2 -23100.059} C_VEL
LIN {X 0,Y 184.417,Z 431.289,A -85,B 0,C 180,E1 -23101.63,E2 -23101.63} C_VEL
LIN {X 0,Y 182.463,Z 439.458,A -85,B 0,C 180,E1 -23103.091,E2 -23103.091} C_VEL
LIN {X 0,Y 180.301,Z 447.5,A -85,B 0,C 180,E1 -23104.92,E2 -23104.92} C_VEL
LIN {X 0,Y 178.288,Z 454.142,A -85,B 0,C 180,E1 -23106.785,E2 -23106.785} C_VEL
LIN {X 0,Y 176.2,Z 460.446,A -85,B 0,C 180,E1 -23108.963,E2 -23108.963} C_VEL
LIN {X 0,Y 175.393,Z 462.945,A -85,B 0,C 180,E1 -23109.945,E2 -23109.945} C_VEL
LIN {X 0,Y 173.595,Z 466.457,A -85,B 0,C 180,E1 -23111.393,E2 -23111.393} C_VEL
LIN {X 0,Y 169.076,Z 471.435,A -85,B 0,C 180,E1 -23113.837,E2 -23113.837} C_VEL
LIN {X 0,Y 164.778,Z 475.465,A -85,B 0,C 180,E1 -23116.586,E2 -23116.586} C_VEL
LIN {X 0,Y 163.372,Z 477.481,A -85,B 0,C 180,E1 -23118.468,E2 -23118.468} C_VEL
LIN {X 0,Y 162.879,Z 478.975,A -85,B 0,C 180,E1 -23120.062,E2 -23120.062} C_VEL
LIN {X 0,Y 162.31,Z 480.706,A -85,B 0,C 180,E1 -23122.536,E2 -23122.536} C_VEL
LIN {X 0,Y 161.939,Z 481.943,A -85,B 0,C 180,E1 -23125.021,E2 -23125.021} C_VEL
LIN {X 0,Y 161.796,Z 482.711,A -85,B 0,C 180,E1 -23127.51,E2 -23127.51} C_VEL
LIN {X 0,Y 161.772,Z 483,A -85,B 0,C 180,E1 -23130,E2 -23130} C_VEL
LIN {X 0,Y 161.796,Z 482.7,A -85,B 0,C 180,E1 -23132.49,E2 -23132.49} C_VEL
LIN {X 0,Y 161.935,Z 481.912,A -85,B 0,C 180,E1 -23134.979,E2 -23134.979} C_VEL
LIN {X 0,Y 162.265,Z 480.653,A -85,B 0,C 180,E1 -23137.466,E2 -23137.466} C_VEL
LIN {X 0,Y 163.248,Z 477.749,A -85,B 0,C 180,E1 -23141.17,E2 -23141.17} C_VEL
LIN {X 0,Y 164.204,Z 475.101,A -85,B 0,C 180,E1 -23143.615,E2 -23143.615} C_VEL
LIN {X 0,Y 166.089,Z 469.925,A -85,B 0,C 180,E1 -23147.229,E2 -23147.229} C_VEL
LIN {X 0,Y 168.635,Z 463.095,A -85,B 0,C 180,E1 -23150.747,E2 -23150.747} C_VEL
LIN {X 0,Y 171.247,Z 455.631,A -85,B 0,C 180,E1 -23153.586,E2 -23153.586} C_VEL
LIN {X 0,Y 173.58,Z 448.267,A -85,B 0,C 180,E1 -23155.801,E2 -23155.801} C_VEL
LIN {X 0,Y 175.843,Z 440.376,A -85,B 0,C 180,E1 -23157.685,E2 -23157.685} C_VEL
LIN {X 0,Y 178.248,Z 430.528,A -85,B 0,C 180,E1 -23159.528,E2 -23159.528} C_VEL
LIN {X 0,Y 180.315,Z 419.523,A -85,B 0,C 180,E1 -23161.022,E2 -23161.022} C_VEL
LIN {X 0,Y 181.744,Z 409.82,A -85,B 0,C 180,E1 -23161.94,E2 -23161.94} C_VEL
LIN {X 0,Y 182.687,Z 400.511,A -85,B 0,C 180,E1 -23162.54,E2 -23162.54} C_VEL
LIN {X 0,Y 184.074,Z 370.075,A -85,B 0,C 180,E1 -23163.734,E2 -23163.734} C_VEL
LIN {X 0,Y 183.053,Z 363.735,A -85,B 0,C 180,E1 -23164.242,E2 -23164.242} C_VEL
LIN {X 0,Y 177.836,Z 350.377,A -85,B 0,C 180,E1 -23166.044,E2 -23166.044} C_VEL
LIN {X 0,Y 172.58,Z 339.349,A -85,B 0,C 180,E1 -23167.89,E2 -23167.89} C_VEL
LIN {X 0,Y 168.92,Z 332.962,A -85,B 0,C 180,E1 -23169.204,E2 -23169.204} C_VEL
LIN {X 0,Y 166.357,Z 328.987,A -85,B 0,C 180,E1 -23170.147,E2 -23170.147} C_VEL
LIN {X 0,Y 164.736,Z 326.499,A -85,B 0,C 180,E1 -23170.779,E2 -23170.779} C_VEL
LIN {X 0,Y 164.349,Z 325.208,A -85,B 0,C 180,E1 -23171.207,E2 -23171.207} C_VEL
LIN {X 0,Y 164.281,Z 324.789,A -85,B 0,C 180,E1 -23172.251,E2 -23172.251} C_VEL
LIN {X 0,Y 164.257,Z 324.819,A -85,B 0,C 180,E1 -23176.797,E2 -23176.797} C_VEL
LIN {X 0,Y 164.285,Z 324.764,A -85,B 0,C 180,E1 -23180.355,E2 -23180.355} C_VEL
LIN {X 0,Y 164.322,Z 324.796,A -85,B 0,C 180,E1 -23184.351,E2 -23184.351} C_VEL
LIN {X 0,Y 164.366,Z 324.805,A -85,B 0,C 180,E1 -23189.13,E2 -23189.13} C_VEL
LIN {X 0,Y 164.382,Z 324.819,A -85,B 0,C 180,E1 -23194.689,E2 -23194.689} C_VEL
LIN {X 0,Y 164.412,Z 324.807,A -85,B 0,C 180,E1 -23200.118,E2 -23200.118} C_VEL
LIN {X 0,Y 164.465,Z 324.784,A -85,B 0,C 180,E1 -23205.144,E2 -23205.144} C_VEL
LIN {X 0,Y 164.76,Z 324.772,A -85,B 0,C 180,E1 -23210.176,E2 -23210.176} C_VEL
LIN {X 0,Y 164.814,Z 324.754,A -85,B 0,C 180,E1 -23212.651,E2 -23212.651} C_VEL
LIN {X 0,Y 165.267,Z 324.713,A -85,B 0,C 180,E1 -23220,E2 -23220} C_VEL
LIN {X 0,Y 164.81,Z 324.754,A -85,B 0,C 180,E1 -23227.35,E2 -23227.35} C_VEL
LIN {X 0,Y 164.697,Z 324.771,A -85,B 0,C 180,E1 -23231.056,E2 -23231.056} C_VEL
LIN {X 0,Y 164.423,Z 324.814,A -85,B 0,C 180,E1 -23237.41,E2 -23237.41} C_VEL
LIN {X 0,Y 164.416,Z 324.805,A -85,B 0,C 180,E1 -23239.997,E2 -23239.997} C_VEL
LIN {X 0,Y 164.36,Z 324.825,A -85,B 0,C 180,E1 -23246.112,E2 -23246.112} C_VEL
LIN {X 0,Y 164.354,Z 324.809,A -85,B 0,C 180,E1 -23251.218,E2 -23251.218} C_VEL
LIN {X 0,Y 164.277,Z 324.781,A -85,B 0,C 180,E1 -23256.794,E2 -23256.794} C_VEL
LIN {X 0,Y 164.283,Z 324.765,A -85,B 0,C 180,E1 -23259.919,E2 -23259.919} C_VEL
LIN {X 0,Y 164.278,Z 324.819,A -85,B 0,C 180,E1 -23263.343,E2 -23263.343} C_VEL
LIN {X 0,Y 164.321,Z 324.939,A -85,B 0,C 180,E1 -23268.572,E2 -23268.572} C_VEL
LIN {X 0,Y 164.515,Z 325.895,A -85,B 0,C 180,E1 -23269.136,E2 -23269.136} C_VEL
LIN {X 0,Y 165.987,Z 328.629,A -85,B 0,C 180,E1 -23269.77,E2 -23269.77} C_VEL
LIN {X 0,Y 167.226,Z 330.266,A -85,B 0,C 180,E1 -23270.219,E2 -23270.219} C_VEL
LIN {X 0,Y 171.643,Z 337.499,A -85,B 0,C 180,E1 -23271.815,E2 -23271.815} C_VEL
LIN {X 0,Y 176.974,Z 348.571,A -85,B 0,C 180,E1 -23273.709,E2 -23273.709} C_VEL
LIN {X 0,Y 182.93,Z 363.208,A -85,B 0,C 180,E1 -23275.753,E2 -23275.753} C_VEL
LIN {X 0,Y 183.594,Z 366.327,A -85,B 0,C 180,E1 -23276.038,E2 -23276.038} C_VEL
LIN {X 0,Y 184.105,Z 371.672,A -85,B 0,C 180,E1 -23276.391,E2 -23276.391} C_VEL
LIN {X 0,Y 182.639,Z 400.884,A -85,B 0,C 180,E1 -23277.519,E2 -23277.519} C_VEL
LIN {X 0,Y 181.444,Z 412.081,A -85,B 0,C 180,E1 -23278.269,E2 -23278.269} C_VEL
LIN {X 0,Y 179.565,Z 423.861,A -85,B 0,C 180,E1 -23279.563,E2 -23279.563} C_VEL
LIN {X 0,Y 177.912,Z 432.075,A -85,B 0,C 180,E1 -23280.791,E2 -23280.791} C_VEL
LIN {X 0,Y 175.872,Z 440.205,A -85,B 0,C 180,E1 -23282.32,E2 -23282.32} C_VEL
LIN {X 0,Y 173.631,Z 448.124,A -85,B 0,C 180,E1 -23284.208,E2 -23284.208} C_VEL
LIN {X 0,Y 171.287,Z 455.511,A -85,B 0,C 180,E1 -23286.419,E2 -23286.419} C_VEL
LIN {X 0,Y 168.664,Z 462.997,A -85,B 0,C 180,E1 -23289.257,E2 -23289.257} C_VEL
LIN {X 0,Y 166.143,Z 469.857,A -85,B 0,C 180,E1 -23292.776,E2 -23292.776} C_VEL
LIN {X 0,Y 164.235,Z 475.047,A -85,B 0,C 180,E1 -23296.388,E2 -23296.388} C_VEL
LIN {X 0,Y 163.265,Z 477.708,A -85,B 0,C 180,E1 -23298.831,E2 -23298.831} C_VEL
LIN {X 0,Y 162.267,Z 480.624,A -85,B 0,C 180,E1 -23302.534,E2 -23302.534} C_VEL
LIN {X 0,Y 161.937,Z 481.895,A -85,B 0,C 180,E1 -23305.021,E2 -23305.021} C_VEL
LIN {X 0,Y 161.797,Z 482.694,A -85,B 0,C 180,E1 -23307.511,E2 -23307.511} C_VEL
LIN {X 0,Y 161.773,Z 482.999,A -85,B 0,C 180,E1 -23310,E2 -23310} C_VEL
LIN {X 0,Y 161.797,Z 482.716,A -85,B 0,C 180,E1 -23312.489,E2 -23312.489} C_VEL
LIN {X 0,Y 161.937,Z 481.961,A -85,B 0,C 180,E1 -23314.979,E2 -23314.979} C_VEL
LIN {X 0,Y 162.266,Z 480.735,A -85,B 0,C 180,E1 -23317.466,E2 -23317.466} C_VEL
LIN {X 0,Y 163.248,Z 477.865,A -85,B 0,C 180,E1 -23321.17,E2 -23321.17} C_VEL
LIN {X 0,Y 164.193,Z 475.252,A -85,B 0,C 180,E1 -23323.616,E2 -23323.616} C_VEL
LIN {X 0,Y 166.095,Z 470.118,A -85,B 0,C 180,E1 -23327.229,E2 -23327.229} C_VEL
LIN {X 0,Y 168.146,Z 464.596,A -85,B 0,C 180,E1 -23330.171,E2 -23330.171} C_VEL
LIN {X 0,Y 170.64,Z 457.654,A -85,B 0,C 180,E1 -23333.033,E2 -23333.033} C_VEL
LIN {X 0,Y 173.268,Z 449.687,A -85,B 0,C 180,E1 -23335.528,E2 -23335.528} C_VEL
LIN {X 0,Y 175.513,Z 442.091,A -85,B 0,C 180,E1 -23337.418,E2 -23337.418} C_VEL
LIN {X 0,Y 177.528,Z 434.342,A -85,B 0,C 180,E1 -23338.962,E2 -23338.962} C_VEL
LIN {X 0,Y 179.28,Z 426.371,A -85,B 0,C 180,E1 -23340.229,E2 -23340.229} C_VEL
LIN {X 0,Y 180.764,Z 417.545,A -85,B 0,C 180,E1 -23341.331,E2 -23341.331} C_VEL
LIN {X 0,Y 181.974,Z 408.482,A -85,B 0,C 180,E1 -23342.156,E2 -23342.156} C_VEL
LIN {X 0,Y 182.826,Z 399.241,A -85,B 0,C 180,E1 -23342.722,E2 -23342.722} C_VEL
LIN {X 0,Y 184.23,Z 370.653,A -85,B 0,C 180,E1 -23343.806,E2 -23343.806} C_VEL
LIN {X 0,Y 183.176,Z 363.771,A -85,B 0,C 180,E1 -23344.346,E2 -23344.346} C_VEL
LIN {X 0,Y 177.518,Z 349.561,A -85,B 0,C 180,E1 -23346.298,E2 -23346.298} C_VEL
LIN {X 0,Y 171.371,Z 336.915,A -85,B 0,C 180,E1 -23348.481,E2 -23348.481} C_VEL
LIN {X 0,Y 168.506,Z 332.411,A -85,B 0,C 180,E1 -23349.502,E2 -23349.502} C_VEL
LIN {X 0,Y 166.41,Z 329.054,A -85,B 0,C 180,E1 -23350.285,E2 -23350.285} C_VEL
LIN {X 0,Y 164.781,Z 326.647,A -85,B 0,C 180,E1 -23350.913,E2 -23350.913} C_VEL
LIN {X 0,Y 164.355,Z 325.288,A -85,B 0,C 180,E1 -23351.325,E2 -23351.325} C_VEL
LIN {X 0,Y 164.297,Z 324.855,A -85,B 0,C 180,E1 -23351.781,E2 -23351.781} C_VEL
LIN {X 0,Y 164.258,Z 324.822,A -85,B 0,C 180,E1 -23356.797,E2 -23356.797} C_VEL
LIN {X 0,Y 164.285,Z 324.765,A -85,B 0,C 180,E1 -23360.355,E2 -23360.355} C_VEL
LIN {X 0,Y 164.323,Z 324.793,A -85,B 0,C 180,E1 -23364.351,E2 -23364.351} C_VEL
LIN {X 0,Y 164.367,Z 324.806,A -85,B 0,C 180,E1 -23369.129,E2 -23369.129} C_VEL
LIN {X 0,Y 164.382,Z 324.819,A -85,B 0,C 180,E1 -23374.688,E2 -23374.688} C_VEL
LIN {X 0,Y 164.413,Z 324.806,A -85,B 0,C 180,E1 -23380.117,E2 -23380.117} C_VEL
LIN {X 0,Y 164.466,Z 324.784,A -85,B 0,C 180,E1 -23385.144,E2 -23385.144} C_VEL
LIN {X 0,Y 164.76,Z 324.772,A -85,B 0,C 180,E1 -23390.176,E2 -23390.176} C_VEL
LIN {X 0,Y 164.815,Z 324.755,A -85,B 0,C 180,E1 -23392.65,E2 -23392.65} C_VEL
LIN {X 0,Y 165.267,Z 324.712,A -85,B 0,C 180,E1 -23400,E2 -23400} C_VEL
LIN {X 0,Y 164.81,Z 324.755,A -85,B 0,C 180,E1 -23407.35,E2 -23407.35} C_VEL
LIN {X 0,Y 164.697,Z 324.771,A -85,B 0,C 180,E1 -23411.055,E2 -23411.055} C_VEL
LIN {X 0,Y 164.423,Z 324.814,A -85,B 0,C 180,E1 -23417.41,E2 -23417.41} C_VEL
LIN {X 0,Y 164.416,Z 324.804,A -85,B 0,C 180,E1 -23419.996,E2 -23419.996} C_VEL
LIN {X 0,Y 164.359,Z 324.825,A -85,B 0,C 180,E1 -23426.112,E2 -23426.112} C_VEL
LIN {X 0,Y 164.353,Z 324.81,A -85,B 0,C 180,E1 -23431.217,E2 -23431.217} C_VEL
LIN {X 0,Y 164.276,Z 324.78,A -85,B 0,C 180,E1 -23436.794,E2 -23436.794} C_VEL
LIN {X 0,Y 164.282,Z 324.766,A -85,B 0,C 180,E1 -23439.918,E2 -23439.918} C_VEL
LIN {X 0,Y 164.277,Z 324.822,A -85,B 0,C 180,E1 -23443.342,E2 -23443.342} C_VEL
LIN {X 0,Y 164.319,Z 324.981,A -85,B 0,C 180,E1 -23448.457,E2 -23448.457} C_VEL
LIN {X 0,Y 164.61,Z 326.155,A -85,B 0,C 180,E1 -23449.038,E2 -23449.038} C_VEL
LIN {X 0,Y 166.192,Z 328.866,A -85,B 0,C 180,E1 -23449.686,E2 -23449.686} C_VEL
LIN {X 0,Y 167.334,Z 330.501,A -85,B 0,C 180,E1 -23450.107,E2 -23450.107} C_VEL
LIN {X 0,Y 171.348,Z 336.898,A -85,B 0,C 180,E1 -23451.557,E2 -23451.557} C_VEL
LIN {X 0,Y 177.312,Z 349.177,A -85,B 0,C 180,E1 -23453.679,E2 -23453.679} C_VEL
LIN {X 0,Y 182.187,Z 361.202,A -85,B 0,C 180,E1 -23455.366,E2 -23455.366} C_VEL
LIN {X 0,Y 183.6,Z 365.577,A -85,B 0,C 180,E1 -23455.873,E2 -23455.873} C_VEL
LIN {X 0,Y 184.256,Z 371.348,A -85,B 0,C 180,E1 -23456.276,E2 -23456.276} C_VEL
LIN {X 0,Y 182.733,Z 401.123,A -85,B 0,C 180,E1 -23457.423,E2 -23457.423} C_VEL
LIN {X 0,Y 181.562,Z 412.171,A -85,B 0,C 180,E1 -23458.172,E2 -23458.172} C_VEL
LIN {X 0,Y 179.684,Z 423.761,A -85,B 0,C 180,E1 -23459.439,E2 -23459.439} C_VEL
LIN {X 0,Y 177.798,Z 433.027,A -85,B 0,C 180,E1 -23460.847,E2 -23460.847} C_VEL
LIN {X 0,Y 175.825,Z 440.691,A -85,B 0,C 180,E1 -23462.312,E2 -23462.312} C_VEL
LIN {X 0,Y 173.6,Z 448.523,A -85,B 0,C 180,E1 -23464.203,E2 -23464.203} C_VEL
LIN {X 0,Y 171.226,Z 455.848,A -85,B 0,C 180,E1 -23466.411,E2 -23466.411} C_VEL
LIN {X 0,Y 168.636,Z 463.276,A -85,B 0,C 180,E1 -23469.254,E2 -23469.254} C_VEL
LIN {X 0,Y 166.099,Z 470.05,A -85,B 0,C 180,E1 -23472.772,E2 -23472.772} C_VEL
LIN {X 0,Y 164.209,Z 475.198,A -85,B 0,C 180,E1 -23476.385,E2 -23476.385} C_VEL
LIN {X 0,Y 163.372,Z 477.481,A -85,B 0,C 180,E1 -23478.468,E2 -23478.468} C_VEL
LIN {X 0,Y 162.104,Z 479.313,A -85,B 0,C 180,E1 -23480.41,E2 -23480.41} C_VEL
LIN {X 0,Y 158.547,Z 481.453,A -85,B 0,C 180,E1 -23483.631,E2 -23483.631} C_VEL
LIN {X 0,Y 155.339,Z 482.666,A -85,B 0,C 180,E1 -23487.045,E2 -23487.045} C_VEL
LIN {X 0,Y 154.653,Z 482.925,A -85,B 0,C 180,E1 -23489.222,E2 -23489.222} C_VEL
LIN {X 0,Y 154.699,Z 482.7,A -85,B 0,C 180,E1 -23492.604,E2 -23492.604} C_VEL
LIN {X 0,Y 154.86,Z 481.912,A -85,B 0,C 180,E1 -23495.208,E2 -23495.208} C_VEL
LIN {X 0,Y 155.223,Z 480.652,A -85,B 0,C 180,E1 -23497.806,E2 -23497.806} C_VEL
LIN {X 0,Y 156.291,Z 477.749,A -85,B 0,C 180,E1 -23501.674,E2 -23501.674} C_VEL
LIN {X 0,Y 157.302,Z 475.1,A -85,B 0,C 180,E1 -23504.225,E2 -23504.225} C_VEL
LIN {X 0,Y 159.327,Z 469.923,A -85,B 0,C 180,E1 -23507.985,E2 -23507.985} C_VEL
LIN {X 0,Y 162.015,Z 463.093,A -85,B 0,C 180,E1 -23511.636,E2 -23511.636} C_VEL
LIN {X 0,Y 164.759,Z 455.628,A -85,B 0,C 180,E1 -23514.575,E2 -23514.575} C_VEL
LIN {X 0,Y 167.227,Z 448.264,A -85,B 0,C 180,E1 -23516.858,E2 -23516.858} C_VEL
LIN {X 0,Y 169.58,Z 440.372,A -85,B 0,C 180,E1 -23518.801,E2 -23518.801} C_VEL
LIN {X 0,Y 171.725,Z 432.028,A -85,B 0,C 180,E1 -23520.427,E2 -23520.427} C_VEL
LIN {X 0,Y 173.943,Z 421.437,A -85,B 0,C 180,E1 -23522.009,E2 -23522.009} C_VEL
LIN {X 0,Y 175.686,Z 410.508,A -85,B 0,C 180,E1 -23523.109,E2 -23523.109} C_VEL
LIN {X 0,Y 176.738,Z 400.743,A -85,B 0,C 180,E1 -23523.763,E2 -23523.763} C_VEL
LIN {X 0,Y 178.192,Z 371.193,A -85,B 0,C 180,E1 -23524.952,E2 -23524.952} C_VEL
LIN {X 0,Y 177.309,Z 365.922,A -85,B 0,C 180,E1 -23525.407,E2 -23525.407} C_VEL
LIN {X 0,Y 172.228,Z 353.048,A -85,B 0,C 180,E1 -23527.275,E2 -23527.275} C_VEL
LIN {X 0,Y 167.214,Z 342.406,A -85,B 0,C 180,E1 -23529.168,E2 -23529.168} C_VEL
LIN {X 0,Y 164.232,Z 337.348,A -85,B 0,C 180,E1 -23530.303,E2 -23530.303} C_VEL
LIN {X 0,Y 160.239,Z 331.035,A -85,B 0,C 180,E1 -23531.896,E2 -23531.896} C_VEL
LIN {X 0,Y 157.787,Z 327.666,A -85,B 0,C 180,E1 -23532.911,E2 -23532.911} C_VEL
LIN {X 0,Y 157.332,Z 326.175,A -85,B 0,C 180,E1 -23533.372,E2 -23533.372} C_VEL
LIN {X 0,Y 157.178,Z 325.703,A -85,B 0,C 180,E1 -23534.323,E2 -23534.323} C_VEL
LIN {X 0,Y 157.19,Z 325.65,A -85,B 0,C 180,E1 -23539.469,E2 -23539.469} C_VEL
LIN {X 0,Y 157.27,Z 325.673,A -85,B 0,C 180,E1 -23544.484,E2 -23544.484} C_VEL
LIN {X 0,Y 157.279,Z 325.697,A -85,B 0,C 180,E1 -23548.102,E2 -23548.102} C_VEL
LIN {X 0,Y 157.306,Z 325.703,A -85,B 0,C 180,E1 -23553.464,E2 -23553.464} C_VEL
LIN {X 0,Y 157.356,Z 325.679,A -85,B 0,C 180,E1 -23559.702,E2 -23559.702} C_VEL
LIN {X 0,Y 157.4,Z 325.668,A -85,B 0,C 180,E1 -23564.461,E2 -23564.461} C_VEL
LIN {X 0,Y 157.683,Z 325.652,A -85,B 0,C 180,E1 -23569.731,E2 -23569.731} C_VEL
LIN {X 0,Y 157.753,Z 325.637,A -85,B 0,C 180,E1 -23572.32,E2 -23572.32} C_VEL
LIN {X 0,Y 158.229,Z 325.589,A -85,B 0,C 180,E1 -23580,E2 -23580} C_VEL
LIN {X 0,Y 157.749,Z 325.637,A -85,B 0,C 180,E1 -23587.681,E2 -23587.681} C_VEL
LIN {X 0,Y 157.626,Z 325.65,A -85,B 0,C 180,E1 -23591.222,E2 -23591.222} C_VEL
LIN {X 0,Y 157.4,Z 325.668,A -85,B 0,C 180,E1 -23595.54,E2 -23595.54} C_VEL
LIN {X 0,Y 157.303,Z 325.68,A -85,B 0,C 180,E1 -23600.942,E2 -23600.942} C_VEL
LIN {X 0,Y 157.289,Z 325.705,A -85,B 0,C 180,E1 -23606.669,E2 -23606.669} C_VEL
LIN {X 0,Y 157.265,Z 325.705,A -85,B 0,C 180,E1 -23612.43,E2 -23612.43} C_VEL
LIN {X 0,Y 157.256,Z 325.658,A -85,B 0,C 180,E1 -23616.445,E2 -23616.445} C_VEL
LIN {X 0,Y 157.187,Z 325.671,A -85,B 0,C 180,E1 -23622.119,E2 -23622.119} C_VEL
LIN {X 0,Y 157.256,Z 325.875,A -85,B 0,C 180,E1 -23626.4,E2 -23626.4} C_VEL
LIN {X 0,Y 157.475,Z 326.897,A -85,B 0,C 180,E1 -23626.948,E2 -23626.948} C_VEL
LIN {X 0,Y 159.094,Z 329.715,A -85,B 0,C 180,E1 -23627.7,E2 -23627.7} C_VEL
LIN {X 0,Y 160.185,Z 330.933,A -85,B 0,C 180,E1 -23628.126,E2 -23628.126} C_VEL
LIN {X 0,Y 162.5,Z 334.485,A -85,B 0,C 180,E1 -23629.058,E2 -23629.058} C_VEL
LIN {X 0,Y 166.793,Z 341.532,A -85,B 0,C 180,E1 -23630.711,E2 -23630.711} C_VEL
LIN {X 0,Y 171.929,Z 352.388,A -85,B 0,C 180,E1 -23632.66,E2 -23632.66} C_VEL
LIN {X 0,Y 177.558,Z 366.553,A -85,B 0,C 180,E1 -23634.725,E2 -23634.725} C_VEL
LIN {X 0,Y 178.208,Z 372.605,A -85,B 0,C 180,E1 -23635.165,E2 -23635.165} C_VEL
LIN {X 0,Y 176.749,Z 400.388,A -85,B 0,C 180,E1 -23636.261,E2 -23636.261} C_VEL
LIN {X 0,Y 175.652,Z 410.365,A -85,B 0,C 180,E1 -23636.915,E2 -23636.915} C_VEL
LIN {X 0,Y 174.007,Z 421.39,A -85,B 0,C 180,E1 -23638.042,E2 -23638.042} C_VEL
LIN {X 0,Y 171.665,Z 432.436,A -85,B 0,C 180,E1 -23639.699,E2 -23639.699} C_VEL
LIN {X 0,Y 169.625,Z 440.209,A -85,B 0,C 180,E1 -23641.207,E2 -23641.207} C_VEL
LIN {X 0,Y 167.27,Z 448.127,A -85,B 0,C 180,E1 -23643.15,E2 -23643.15} C_VEL
LIN {X 0,Y 164.79,Z 455.514,A -85,B 0,C 180,E1 -23645.43,E2 -23645.43} C_VEL
LIN {X 0,Y 162.045,Z 462.999,A -85,B 0,C 180,E1 -23648.368,E2 -23648.368} C_VEL
LIN {X 0,Y 159.368,Z 469.859,A -85,B 0,C 180,E1 -23652.02,E2 -23652.02} C_VEL
LIN {X 0,Y 157.332,Z 475.048,A -85,B 0,C 180,E1 -23655.778,E2 -23655.778} C_VEL
LIN {X 0,Y 156.308,Z 477.709,A -85,B 0,C 180,E1 -23658.327,E2 -23658.327} C_VEL
LIN {X 0,Y 155.225,Z 480.625,A -85,B 0,C 180,E1 -23662.194,E2 -23662.194} C_VEL
LIN {X 0,Y 154.862,Z 481.895,A -85,B 0,C 180,E1 -23664.793,E2 -23664.793} C_VEL
LIN {X 0,Y 154.657,Z 482.855,A -85,B 0,C 180,E1 -23668.699,E2 -23668.699} C_VEL
LIN {X 0,Y 154.649,Z 482.893,A -85,B 0,C 180,E1 -23671.172,E2 -23671.172} C_VEL
LIN {X 0,Y 154.862,Z 481.96,A -85,B 0,C 180,E1 -23675.207,E2 -23675.207} C_VEL
LIN {X 0,Y 155.225,Z 480.734,A -85,B 0,C 180,E1 -23677.806,E2 -23677.806} C_VEL
LIN {X 0,Y 156.291,Z 477.864,A -85,B 0,C 180,E1 -23681.674,E2 -23681.674} C_VEL
LIN {X 0,Y 157.277,Z 475.251,A -85,B 0,C 180,E1 -23684.227,E2 -23684.227} C_VEL
LIN {X 0,Y 159.331,Z 470.116,A -85,B 0,C 180,E1 -23687.984,E2 -23687.984} C_VEL
LIN {X 0,Y 161.5,Z 464.594,A -85,B 0,C 180,E1 -23691.039,E2 -23691.039} C_VEL
LIN {X 0,Y 164.139,Z 457.651,A -85,B 0,C 180,E1 -23694.001,E2 -23694.001} C_VEL
LIN {X 0,Y 166.895,Z 449.683,A -85,B 0,C 180,E1 -23696.578,E2 -23696.578} C_VEL
LIN {X 0,Y 169.241,Z 442.087,A -85,B 0,C 180,E1 -23698.525,E2 -23698.525} C_VEL
LIN {X 0,Y 171.301,Z 434.592,A -85,B 0,C 180,E1 -23700.064,E2 -23700.064} C_VEL
LIN {X 0,Y 173.172,Z 426.365,A -85,B 0,C 180,E1 -23701.414,E2 -23701.414} C_VEL
LIN {X 0,Y 174.728,Z 417.556,A -85,B 0,C 180,E1 -23702.541,E2 -23702.541} C_VEL
LIN {X 0,Y 175.997,Z 408.526,A -85,B 0,C 180,E1 -23703.382,E2 -23703.382} C_VEL
LIN {X 0,Y 176.909,Z 399.224,A -85,B 0,C 180,E1 -23703.962,E2 -23703.962} C_VEL
LIN {X 0,Y 178.315,Z 371.369,A -85,B 0,C 180,E1 -23705.052,E2 -23705.052} C_VEL
LIN {X 0,Y 177.571,Z 366.557,A -85,B 0,C 180,E1 -23705.454,E2 -23705.454} C_VEL
LIN {X 0,Y 172.471,Z 353.407,A -85,B 0,C 180,E1 -23707.341,E2 -23707.341} C_VEL
LIN {X 0,Y 166.767,Z 341.435,A -85,B 0,C 180,E1 -23709.501,E2 -23709.501} C_VEL
LIN {X 0,Y 162.105,Z 334.019,A -85,B 0,C 180,E1 -23711.299,E2 -23711.299} C_VEL
LIN {X 0,Y 159.52,Z 330.05,A -85,B 0,C 180,E1 -23712.355,E2 -23712.355} C_VEL
LIN {X 0,Y 157.699,Z 327.485,A -85,B 0,C 180,E1 -23713.13,E2 -23713.13} C_VEL
LIN {X 0,Y 157.293,Z 326.095,A -85,B 0,C 180,E1 -23713.61,E2 -23713.61} C_VEL
LIN {X 0,Y 157.181,Z 325.724,A -85,B 0,C 180,E1 -23714.323,E2 -23714.323} C_VEL
LIN {X 0,Y 157.19,Z 325.652,A -85,B 0,C 180,E1 -23719.469,E2 -23719.469} C_VEL
LIN {X 0,Y 157.271,Z 325.67,A -85,B 0,C 180,E1 -23724.483,E2 -23724.483} C_VEL
LIN {X 0,Y 157.28,Z 325.698,A -85,B 0,C 180,E1 -23728.102,E2 -23728.102} C_VEL
LIN {X 0,Y 157.307,Z 325.703,A -85,B 0,C 180,E1 -23733.463,E2 -23733.463} C_VEL
LIN {X 0,Y 157.356,Z 325.678,A -85,B 0,C 180,E1 -23739.702,E2 -23739.702} C_VEL
LIN {X 0,Y 157.4,Z 325.669,A -85,B 0,C 180,E1 -23744.46,E2 -23744.46} C_VEL
LIN {X 0,Y 157.683,Z 325.652,A -85,B 0,C 180,E1 -23749.73,E2 -23749.73} C_VEL
LIN {X 0,Y 157.753,Z 325.638,A -85,B 0,C 180,E1 -23752.319,E2 -23752.319} C_VEL
LIN {X 0,Y 158.229,Z 325.589,A -85,B 0,C 180,E1 -23760,E2 -23760} C_VEL
LIN {X 0,Y 157.749,Z 325.638,A -85,B 0,C 180,E1 -23767.681,E2 -23767.681} C_VEL
LIN {X 0,Y 157.626,Z 325.649,A -85,B 0,C 180,E1 -23771.221,E2 -23771.221} C_VEL
LIN {X 0,Y 157.4,Z 325.668,A -85,B 0,C 180,E1 -23775.539,E2 -23775.539} C_VEL
LIN {X 0,Y 157.303,Z 325.679,A -85,B 0,C 180,E1 -23780.942,E2 -23780.942} C_VEL
LIN {X 0,Y 157.289,Z 325.704,A -85,B 0,C 180,E1 -23786.668,E2 -23786.668} C_VEL
LIN {X 0,Y 157.264,Z 325.706,A -85,B 0,C 180,E1 -23792.43,E2 -23792.43} C_VEL
LIN {X 0,Y 157.255,Z 325.656,A -85,B 0,C 180,E1 -23796.444,E2 -23796.444} C_VEL
LIN {X 0,Y 157.186,Z 325.674,A -85,B 0,C 180,E1 -23802.118,E2 -23802.118} C_VEL
LIN {X 0,Y 157.269,Z 325.967,A -85,B 0,C 180,E1 -23806.335,E2 -23806.335} C_VEL
LIN {X 0,Y 157.521,Z 327.026,A -85,B 0,C 180,E1 -23806.81,E2 -23806.81} C_VEL
LIN {X 0,Y 159.188,Z 329.747,A -85,B 0,C 180,E1 -23807.562,E2 -23807.562} C_VEL
LIN {X 0,Y 160.258,Z 331.073,A -85,B 0,C 180,E1 -23807.99,E2 -23807.99} C_VEL
LIN {X 0,Y 162.575,Z 334.569,A -85,B 0,C 180,E1 -23808.923,E2 -23808.923} C_VEL
LIN {X 0,Y 166.976,Z 341.918,A -85,B 0,C 180,E1 -23810.629,E2 -23810.629} C_VEL
LIN {X 0,Y 172.531,Z 353.644,A -85,B 0,C 180,E1 -23812.732,E2 -23812.732} C_VEL
LIN {X 0,Y 176.834,Z 364.468,A -85,B 0,C 180,E1 -23814.318,E2 -23814.318} C_VEL
LIN {X 0,Y 177.922,Z 368.031,A -85,B 0,C 180,E1 -23814.742,E2 -23814.742} C_VEL
LIN {X 0,Y 178.34,Z 372.843,A -85,B 0,C 180,E1 -23815.069,E2 -23815.069} C_VEL
LIN {X 0,Y 176.794,Z 401.139,A -85,B 0,C 180,E1 -23816.185,E2 -23816.185} C_VEL
LIN {X 0,Y 175.617,Z 411.662,A -85,B 0,C 180,E1 -23816.905,E2 -23816.905} C_VEL
LIN {X 0,Y 173.761,Z 423.023,A -85,B 0,C 180,E1 -23818.143,E2 -23818.143} C_VEL
LIN {X 0,Y 171.818,Z 432.28,A -85,B 0,C 180,E1 -23819.559,E2 -23819.559} C_VEL
LIN {X 0,Y 169.567,Z 440.694,A -85,B 0,C 180,E1 -23821.197,E2 -23821.197} C_VEL
LIN {X 0,Y 167.238,Z 448.527,A -85,B 0,C 180,E1 -23823.144,E2 -23823.144} C_VEL
LIN {X 0,Y 164.734,Z 455.85,A -85,B 0,C 180,E1 -23825.421,E2 -23825.421} C_VEL
LIN {X 0,Y 162.016,Z 463.278,A -85,B 0,C 180,E1 -23828.364,E2 -23828.364} C_VEL
LIN {X 0,Y 159.336,Z 470.052,A -85,B 0,C 180,E1 -23832.016,E2 -23832.016} C_VEL
LIN {X 0,Y 157.307,Z 475.199,A -85,B 0,C 180,E1 -23835.776,E2 -23835.776} C_VEL
LIN {X 0,Y 155.876,Z 478.975,A -85,B 0,C 180,E1 -23839.61,E2 -23839.61} C_VEL
LIN {X 0,Y 155.284,Z 480.706,A -85,B 0,C 180,E1 -23842.197,E2 -23842.197} C_VEL
LIN {X 0,Y 154.864,Z 481.944,A -85,B 0,C 180,E1 -23844.793,E2 -23844.793} C_VEL
LIN {X 0,Y 154.648,Z 482.887,A -85,B 0,C 180,E1 -23848.828,E2 -23848.828} C_VEL
LIN {X 0,Y 154.653,Z 482.925,A -85,B 0,C 180,E1 -23849.222,E2 -23849.222} C_VEL
LIN {X 0,Y 154.368,Z 482.965,A -85,B 0,C 180,E1 -23850.673,E2 -23850.673} C_VEL
LIN {X 0,Y 153.087,Z 482.7,A -85,B 0,C 180,E1 -23852.824,E2 -23852.824} C_VEL
LIN {X 0,Y 149.702,Z 481.224,A -85,B 0,C 180,E1 -23857.131,E2 -23857.131} C_VEL
LIN {X 0,Y 148.745,Z 479.497,A -85,B 0,C 180,E1 -23860.099,E2 -23860.099} C_VEL
LIN {X 0,Y 148.883,Z 478.925,A -85,B 0,C 180,E1 -23860.842,E2 -23860.842} C_VEL
LIN {X 0,Y 149.824,Z 476.578,A -85,B 0,C 180,E1 -23863.564,E2 -23863.564} C_VEL
LIN {X 0,Y 151.766,Z 471.835,A -85,B 0,C 180,E1 -23867.517,E2 -23867.517} C_VEL
LIN {X 0,Y 153.9,Z 466.699,A -85,B 0,C 180,E1 -23870.726,E2 -23870.726} C_VEL
LIN {X 0,Y 155.941,Z 461.676,A -85,B 0,C 180,E1 -23873.225,E2 -23873.225} C_VEL
LIN {X 0,Y 158.316,Z 455.626,A -85,B 0,C 180,E1 -23875.646,E2 -23875.646} C_VEL
LIN {X 0,Y 160.923,Z 448.26,A -85,B 0,C 180,E1 -23878,E2 -23878} C_VEL
LIN {X 0,Y 163.382,Z 440.368,A -85,B 0,C 180,E1 -23880.003,E2 -23880.003} C_VEL
LIN {X 0,Y 165.923,Z 431.055,A -85,B 0,C 180,E1 -23881.841,E2 -23881.841} C_VEL
LIN {X 0,Y 168.343,Z 419.396,A -85,B 0,C 180,E1 -23883.522,E2 -23883.522} C_VEL
LIN {X 0,Y 169.955,Z 409.093,A -85,B 0,C 180,E1 -23884.529,E2 -23884.529} C_VEL
LIN {X 0,Y 170.96,Z 399.745,A -85,B 0,C 180,E1 -23885.136,E2 -23885.136} C_VEL
LIN {X 0,Y 172.342,Z 371.844,A -85,B 0,C 180,E1 -23886.289,E2 -23886.289} C_VEL
LIN {X 0,Y 171.639,Z 368.166,A -85,B 0,C 180,E1 -23886.649,E2 -23886.649} C_VEL
LIN {X 0,Y 166.52,Z 355.2,A -85,B 0,C 180,E1 -23888.667,E2 -23888.667} C_VEL
LIN {X 0,Y 161.608,Z 344.894,A -85,B 0,C 180,E1 -23890.662,E2 -23890.662} C_VEL
LIN {X 0,Y 155.397,Z 335.147,A -85,B 0,C 180,E1 -23893.261,E2 -23893.261} C_VEL
LIN {X 0,Y 153.262,Z 331.83,A -85,B 0,C 180,E1 -23894.228,E2 -23894.228} C_VEL
LIN {X 0,Y 150.942,Z 329.089,A -85,B 0,C 180,E1 -23895.272,E2 -23895.272} C_VEL
LIN {X 0,Y 150.232,Z 327.174,A -85,B 0,C 180,E1 -23895.861,E2 -23895.861} C_VEL
LIN {X 0,Y 150.123,Z 326.612,A -85,B 0,C 180,E1 -23896.663,E2 -23896.663} C_VEL
LIN {X 0,Y 150.172,Z 326.525,A -85,B 0,C 180,E1 -23902.71,E2 -23902.71} C_VEL
LIN {X 0,Y 150.205,Z 326.586,A -85,B 0,C 180,E1 -23907.372,E2 -23907.372} C_VEL
LIN {X 0,Y 150.225,Z 326.578,A -85,B 0,C 180,E1 -23912.73,E2 -23912.73} C_VEL
LIN {X 0,Y 150.279,Z 326.555,A -85,B 0,C 180,E1 -23919.277,E2 -23919.277} C_VEL
LIN {X 0,Y 150.306,Z 326.559,A -85,B 0,C 180,E1 -23923.707,E2 -23923.707} C_VEL
LIN {X 0,Y 150.602,Z 326.528,A -85,B 0,C 180,E1 -23929.242,E2 -23929.242} C_VEL
LIN {X 0,Y 150.692,Z 326.519,A -85,B 0,C 180,E1 -23931.957,E2 -23931.957} C_VEL
LIN {X 0,Y 151.19,Z 326.466,A -85,B 0,C 180,E1 -23940,E2 -23940} C_VEL
LIN {X 0,Y 150.673,Z 326.521,A -85,B 0,C 180,E1 -23948.044,E2 -23948.044} C_VEL
LIN {X 0,Y 150.569,Z 326.524,A -85,B 0,C 180,E1 -23951.426,E2 -23951.426} C_VEL
LIN {X 0,Y 150.306,Z 326.559,A -85,B 0,C 180,E1 -23956.293,E2 -23956.293} C_VEL
LIN {X 0,Y 150.28,Z 326.555,A -85,B 0,C 180,E1 -23960.723,E2 -23960.723} C_VEL
LIN {X 0,Y 150.225,Z 326.579,A -85,B 0,C 180,E1 -23967.27,E2 -23967.27} C_VEL
LIN {X 0,Y 150.206,Z 326.585,A -85,B 0,C 180,E1 -23972.629,E2 -23972.629} C_VEL
LIN {X 0,Y 150.166,Z 326.525,A -85,B 0,C 180,E1 -23977.476,E2 -23977.476} C_VEL
LIN {X 0,Y 150.133,Z 326.625,A -85,B 0,C 180,E1 -23983.544,E2 -23983.544} C_VEL
LIN {X 0,Y 150.264,Z 327.219,A -85,B 0,C 180,E1 -23984.234,E2 -23984.234} C_VEL
LIN {X 0,Y 151.521,Z 329.98,A -85,B 0,C 180,E1 -23985.052,E2 -23985.052} C_VEL
LIN {X 0,Y 153.33,Z 331.992,A -85,B 0,C 180,E1 -23985.852,E2 -23985.852} C_VEL
LIN {X 0,Y 155.492,Z 335.345,A -85,B 0,C 180,E1 -23986.829,E2 -23986.829} C_VEL
LIN {X 0,Y 161.619,Z 344.837,A -85,B 0,C 180,E1 -23989.383,E2 -23989.383} C_VEL
LIN {X 0,Y 166.782,Z 355.804,A -85,B 0,C 180,E1 -23991.482,E2 -23991.482} C_VEL
LIN {X 0,Y 172.025,Z 369.259,A -85,B 0,C 180,E1 -23993.548,E2 -23993.548} C_VEL
LIN {X 0,Y 172.38,Z 373.824,A -85,B 0,C 180,E1 -23993.866,E2 -23993.866} C_VEL
LIN {X 0,Y 170.79,Z 401.16,A -85,B 0,C 180,E1 -23994.968,E2 -23994.968} C_VEL
LIN {X 0,Y 169.588,Z 411.783,A -85,B 0,C 180,E1 -23995.721,E2 -23995.721} C_VEL
LIN {X 0,Y 167.677,Z 423.032,A -85,B 0,C 180,E1 -23996.984,E2 -23996.984} C_VEL
LIN {X 0,Y 165.478,Z 432.842,A -85,B 0,C 180,E1 -23998.534,E2 -23998.534} C_VEL
LIN {X 0,Y 163.453,Z 440.213,A -85,B 0,C 180,E1 -24000.011,E2 -24000.011} C_VEL
LIN {X 0,Y 160.973,Z 448.131,A -85,B 0,C 180,E1 -24002.009,E2 -24002.009} C_VEL
LIN {X 0,Y 158.359,Z 455.517,A -85,B 0,C 180,E1 -24004.361,E2 -24004.361} C_VEL
LIN {X 0,Y 155.469,Z 463.001,A -85,B 0,C 180,E1 -24007.404,E2 -24007.404} C_VEL
LIN {X 0,Y 152.633,Z 469.86,A -85,B 0,C 180,E1 -24011.197,E2 -24011.197} C_VEL
LIN {X 0,Y 150.44,Z 475.049,A -85,B 0,C 180,E1 -24015.112,E2 -24015.112} C_VEL
LIN {X 0,Y 149.349,Z 477.71,A -85,B 0,C 180,E1 -24017.775,E2 -24017.775} C_VEL
LIN {X 0,Y 148.206,Z 480.625,A -85,B 0,C 180,E1 -24021.821,E2 -24021.821} C_VEL
LIN {X 0,Y 147.798,Z 481.896,A -85,B 0,C 180,E1 -24024.543,E2 -24024.543} C_VEL
LIN {X 0,Y 147.613,Z 482.695,A -85,B 0,C 180,E1 -24027.271,E2 -24027.271} C_VEL
LIN {X 0,Y 147.589,Z 482.999,A -85,B 0,C 180,E1 -24030,E2 -24030} C_VEL
LIN {X 0,Y 147.613,Z 482.716,A -85,B 0,C 180,E1 -24032.729,E2 -24032.729} C_VEL
LIN {X 0,Y 147.798,Z 481.96,A -85,B 0,C 180,E1 -24035.457,E2 -24035.457} C_VEL
LIN {X 0,Y 148.205,Z 480.733,A -85,B 0,C 180,E1 -24038.179,E2 -24038.179} C_VEL
LIN {X 0,Y 149.327,Z 477.863,A -85,B 0,C 180,E1 -24042.227,E2 -24042.227} C_VEL
LIN {X 0,Y 150.384,Z 475.25,A -85,B 0,C 180,E1 -24044.894,E2 -24044.894} C_VEL
LIN {X 0,Y 152.581,Z 470.115,A -85,B 0,C 180,E1 -24048.809,E2 -24048.809} C_VEL
LIN {X 0,Y 154.898,Z 464.592,A -85,B 0,C 180,E1 -24051.982,E2 -24051.982} C_VEL
LIN {X 0,Y 157.683,Z 457.649,A -85,B 0,C 180,E1 -24055.05,E2 -24055.05} C_VEL
LIN {X 0,Y 160.583,Z 449.68,A -85,B 0,C 180,E1 -24057.71,E2 -24057.71} C_VEL
LIN {X 0,Y 163.036,Z 442.083,A -85,B 0,C 180,E1 -24059.717,E2 -24059.717} C_VEL
LIN {X 0,Y 165.375,Z 433.706,A -85,B 0,C 180,E1 -24061.469,E2 -24061.469} C_VEL
LIN {X 0,Y 167.395,Z 425.234,A -85,B 0,C 180,E1 -24062.844,E2 -24062.844} C_VEL
LIN {X 0,Y 168.911,Z 416.652,A -85,B 0,C 180,E1 -24063.942,E2 -24063.942} C_VEL
LIN {X 0,Y 170.415,Z 406.362,A -85,B 0,C 180,E1 -24064.86,E2 -24064.86} C_VEL
LIN {X 0,Y 171.519,Z 392.193,A -85,B 0,C 180,E1 -24065.602,E2 -24065.602} C_VEL
LIN {X 0,Y 172.461,Z 371.849,A -85,B 0,C 180,E1 -24066.403,E2 -24066.403} C_VEL
LIN {X 0,Y 171.737,Z 368.27,A -85,B 0,C 180,E1 -24066.764,E2 -24066.764} C_VEL
LIN {X 0,Y 166.318,Z 354.454,A -85,B 0,C 180,E1 -24068.918,E2 -24068.918} C_VEL
LIN {X 0,Y 160.899,Z 343.542,A -85,B 0,C 180,E1 -24071.122,E2 -24071.122} C_VEL
LIN {X 0,Y 155.297,Z 335.046,A -85,B 0,C 180,E1 -24073.479,E2 -24073.479} C_VEL
LIN {X 0,Y 152.772,Z 331.261,A -85,B 0,C 180,E1 -24074.627,E2 -24074.627} C_VEL
LIN {X 0,Y 150.912,Z 329.049,A -85,B 0,C 180,E1 -24075.475,E2 -24075.475} C_VEL
LIN {X 0,Y 150.228,Z 327.14,A -85,B 0,C 180,E1 -24076.07,E2 -24076.07} C_VEL
LIN {X 0,Y 150.126,Z 326.587,A -85,B 0,C 180,E1 -24077.081,E2 -24077.081} C_VEL
LIN {X 0,Y 150.173,Z 326.524,A -85,B 0,C 180,E1 -24082.709,E2 -24082.709} C_VEL
LIN {X 0,Y 150.206,Z 326.587,A -85,B 0,C 180,E1 -24087.371,E2 -24087.371} C_VEL
LIN {X 0,Y 150.225,Z 326.576,A -85,B 0,C 180,E1 -24092.73,E2 -24092.73} C_VEL
LIN {X 0,Y 150.28,Z 326.554,A -85,B 0,C 180,E1 -24099.277,E2 -24099.277} C_VEL
LIN {X 0,Y 150.307,Z 326.56,A -85,B 0,C 180,E1 -24103.707,E2 -24103.707} C_VEL
LIN {X 0,Y 150.602,Z 326.527,A -85,B 0,C 180,E1 -24109.242,E2 -24109.242} C_VEL
LIN {X 0,Y 150.692,Z 326.52,A -85,B 0,C 180,E1 -24111.957,E2 -24111.957} C_VEL
LIN {X 0,Y 151.19,Z 326.466,A -85,B 0,C 180,E1 -24120,E2 -24120} C_VEL
LIN {X 0,Y 150.673,Z 326.522,A -85,B 0,C 180,E1 -24128.044,E2 -24128.044} C_VEL
LIN {X 0,Y 150.568,Z 326.524,A -85,B 0,C 180,E1 -24131.425,E2 -24131.425} C_VEL
LIN {X 0,Y 150.306,Z 326.56,A -85,B 0,C 180,E1 -24136.293,E2 -24136.293} C_VEL
LIN {X 0,Y 150.279,Z 326.555,A -85,B 0,C 180,E1 -24140.723,E2 -24140.723} C_VEL
LIN {X 0,Y 150.225,Z 326.577,A -85,B 0,C 180,E1 -24147.27,E2 -24147.27} C_VEL
LIN {X 0,Y 150.205,Z 326.587,A -85,B 0,C 180,E1 -24152.628,E2 -24152.628} C_VEL
LIN {X 0,Y 150.165,Z 326.523,A -85,B 0,C 180,E1 -24157.475,E2 -24157.475} C_VEL
LIN {X 0,Y 150.129,Z 326.632,A -85,B 0,C 180,E1 -24163.44,E2 -24163.44} C_VEL
LIN {X 0,Y 150.281,Z 327.407,A -85,B 0,C 180,E1 -24164.121,E2 -24164.121} C_VEL
LIN {X 0,Y 151.741,Z 330.28,A -85,B 0,C 180,E1 -24164.968,E2 -24164.968} C_VEL
LIN {X 0,Y 153.42,Z 332.122,A -85,B 0,C 180,E1 -24165.711,E2 -24165.711} C_VEL
LIN {X 0,Y 155.72,Z 335.503,A -85,B 0,C 180,E1 -24166.742,E2 -24166.742} C_VEL
LIN {X 0,Y 162.139,Z 345.818,A -85,B 0,C 180,E1 -24169.434,E2 -24169.434} C_VEL
LIN {X 0,Y 167.927,Z 358.322,A -85,B 0,C 180,E1 -24171.776,E2 -24171.776} C_VEL
LIN {X 0,Y 172.2,Z 369.678,A -85,B 0,C 180,E1 -24173.468,E2 -24173.468} C_VEL
LIN {X 0,Y 172.543,Z 373.731,A -85,B 0,C 180,E1 -24173.757,E2 -24173.757} C_VEL
LIN {X 0,Y 170.96,Z 401.155,A -85,B 0,C 180,E1 -24174.864,E2 -24174.864} C_VEL
LIN {X 0,Y 169.554,Z 412.98,A -85,B 0,C 180,E1 -24175.714,E2 -24175.714} C_VEL
LIN {X 0,Y 167.609,Z 423.773,A -85,B 0,C 180,E1 -24176.969,E2 -24176.969} C_VEL
LIN {X 0,Y 165.61,Z 432.781,A -85,B 0,C 180,E1 -24178.406,E2 -24178.406} C_VEL
LIN {X 0,Y 163.381,Z 440.698,A -85,B 0,C 180,E1 -24179.997,E2 -24179.997} C_VEL
LIN {X 0,Y 160.938,Z 448.53,A -85,B 0,C 180,E1 -24182.003,E2 -24182.003} C_VEL
LIN {X 0,Y 158.303,Z 455.853,A -85,B 0,C 180,E1 -24184.351,E2 -24184.351} C_VEL
LIN {X 0,Y 155.438,Z 463.28,A -85,B 0,C 180,E1 -24187.399,E2 -24187.399} C_VEL
LIN {X 0,Y 152.586,Z 470.053,A -85,B 0,C 180,E1 -24191.191,E2 -24191.191} C_VEL
LIN {X 0,Y 150.414,Z 475.2,A -85,B 0,C 180,E1 -24195.109,E2 -24195.109} C_VEL
LIN {X 0,Y 148.899,Z 478.976,A -85,B 0,C 180,E1 -24199.118,E2 -24199.118} C_VEL
LIN {X 0,Y 148.248,Z 480.707,A -85,B 0,C 180,E1 -24201.824,E2 -24201.824} C_VEL
LIN {X 0,Y 147.801,Z 481.944,A -85,B 0,C 180,E1 -24204.543,E2 -24204.543} C_VEL
LIN {X 0,Y 147.612,Z 482.711,A -85,B 0,C 180,E1 -24207.271,E2 -24207.271} C_VEL
LIN {X 0,Y 147.587,Z 483,A -85,B 0,C 180,E1 -24210,E2 -24210} C_VEL
LIN {X 0,Y 147.612,Z 482.7,A -85,B 0,C 180,E1 -24212.729,E2 -24212.729} C_VEL
LIN {X 0,Y 147.796,Z 481.911,A -85,B 0,C 180,E1 -24215.457,E2 -24215.457} C_VEL
LIN {X 0,Y 148.204,Z 480.652,A -85,B 0,C 180,E1 -24218.179,E2 -24218.179} C_VEL
LIN {X 0,Y 148.883,Z 478.925,A -85,B 0,C 180,E1 -24220.842,E2 -24220.842} C_VEL
LIN {X 0,Y 148.982,Z 477.291,A -85,B 0,C 180,E1 -24223.025,E2 -24223.025} C_VEL
LIN {X 0,Y 148.295,Z 475.304,A -85,B 0,C 180,E1 -24225.171,E2 -24225.171} C_VEL
LIN {X 0,Y 146.802,Z 470.321,A -85,B 0,C 180,E1 -24229.353,E2 -24229.353} C_VEL
LIN {X 0,Y 147.086,Z 467.327,A -85,B 0,C 180,E1 -24231.344,E2 -24231.344} C_VEL
LIN {X 0,Y 147.47,Z 466.222,A -85,B 0,C 180,E1 -24231.972,E2 -24231.972} C_VEL
LIN {X 0,Y 150.052,Z 460.257,A -85,B 0,C 180,E1 -24234.931,E2 -24234.931} C_VEL
LIN {X 0,Y 152.622,Z 453.922,A -85,B 0,C 180,E1 -24237.418,E2 -24237.418} C_VEL
LIN {X 0,Y 155.813,Z 445.185,A -85,B 0,C 180,E1 -24240.118,E2 -24240.118} C_VEL
LIN {X 0,Y 158.478,Z 436.517,A -85,B 0,C 180,E1 -24242.151,E2 -24242.151} C_VEL
LIN {X 0,Y 160.842,Z 427.049,A -85,B 0,C 180,E1 -24243.847,E2 -24243.847} C_VEL
LIN {X 0,Y 162.637,Z 418.522,A -85,B 0,C 180,E1 -24244.999,E2 -24244.999} C_VEL
LIN {X 0,Y 164.157,Z 408.989,A -85,B 0,C 180,E1 -24245.945,E2 -24245.945} C_VEL
LIN {X 0,Y 165.204,Z 399.729,A -85,B 0,C 180,E1 -24246.553,E2 -24246.553} C_VEL
LIN {X 0,Y 166.644,Z 372.703,A -85,B 0,C 180,E1 -24247.694,E2 -24247.694} C_VEL
LIN {X 0,Y 164.763,Z 366.935,A -85,B 0,C 180,E1 -24248.514,E2 -24248.514} C_VEL
LIN {X 0,Y 159.87,Z 355.051,A -85,B 0,C 180,E1 -24250.608,E2 -24250.608} C_VEL
LIN {X 0,Y 156.115,Z 347.666,A -85,B 0,C 180,E1 -24252.247,E2 -24252.247} C_VEL
LIN {X 0,Y 151.053,Z 339.817,A -85,B 0,C 180,E1 -24254.525,E2 -24254.525} C_VEL
LIN {X 0,Y 148.663,Z 336.351,A -85,B 0,C 180,E1 -24255.671,E2 -24255.671} C_VEL
LIN {X 0,Y 146.516,Z 333.139,A -85,B 0,C 180,E1 -24256.762,E2 -24256.762} C_VEL
LIN {X 0,Y 145.632,Z 332.054,A -85,B 0,C 180,E1 -24257.209,E2 -24257.209} C_VEL
LIN {X 0,Y 143.772,Z 329.688,A -85,B 0,C 180,E1 -24258.189,E2 -24258.189} C_VEL
LIN {X 0,Y 143.217,Z 328.068,A -85,B 0,C 180,E1 -24258.735,E2 -24258.735} C_VEL
LIN {X 0,Y 143.071,Z 327.458,A -85,B 0,C 180,E1 -24259.667,E2 -24259.667} C_VEL
LIN {X 0,Y 143.078,Z 327.421,A -85,B 0,C 180,E1 -24263.883,E2 -24263.883} C_VEL
LIN {X 0,Y 143.172,Z 327.461,A -85,B 0,C 180,E1 -24267.319,E2 -24267.319} C_VEL
LIN {X 0,Y 143.173,Z 327.447,A -85,B 0,C 180,E1 -24272.074,E2 -24272.074} C_VEL
LIN {X 0,Y 143.217,Z 327.43,A -85,B 0,C 180,E1 -24278.805,E2 -24278.805} C_VEL
LIN {X 0,Y 143.247,Z 327.448,A -85,B 0,C 180,E1 -24282.88,E2 -24282.88} C_VEL
LIN {X 0,Y 143.528,Z 327.4,A -85,B 0,C 180,E1 -24288.705,E2 -24288.705} C_VEL
LIN {X 0,Y 143.615,Z 327.404,A -85,B 0,C 180,E1 -24291.558,E2 -24291.558} C_VEL
LIN {X 0,Y 144.148,Z 327.343,A -85,B 0,C 180,E1 -24300,E2 -24300} C_VEL
LIN {X 0,Y 143.599,Z 327.405,A -85,B 0,C 180,E1 -24308.443,E2 -24308.443} C_VEL
LIN {X 0,Y 143.493,Z 327.401,A -85,B 0,C 180,E1 -24311.611,E2 -24311.611} C_VEL
LIN {X 0,Y 143.247,Z 327.447,A -85,B 0,C 180,E1 -24317.12,E2 -24317.12} C_VEL
LIN {X 0,Y 143.218,Z 327.43,A -85,B 0,C 180,E1 -24321.196,E2 -24321.196} C_VEL
LIN {X 0,Y 143.173,Z 327.448,A -85,B 0,C 180,E1 -24327.926,E2 -24327.926} C_VEL
LIN {X 0,Y 143.156,Z 327.466,A -85,B 0,C 180,E1 -24333.43,E2 -24333.43} C_VEL
LIN {X 0,Y 143.049,Z 327.401,A -85,B 0,C 180,E1 -24339.695,E2 -24339.695} C_VEL
LIN {X 0,Y 143.161,Z 327.815,A -85,B 0,C 180,E1 -24341.121,E2 -24341.121} C_VEL
LIN {X 0,Y 143.567,Z 329.268,A -85,B 0,C 180,E1 -24341.72,E2 -24341.72} C_VEL
LIN {X 0,Y 145.24,Z 331.724,A -85,B 0,C 180,E1 -24342.645,E2 -24342.645} C_VEL
LIN {X 0,Y 146.472,Z 332.993,A -85,B 0,C 180,E1 -24343.255,E2 -24343.255} C_VEL
LIN {X 0,Y 148.469,Z 336.165,A -85,B 0,C 180,E1 -24344.284,E2 -24344.284} C_VEL
LIN {X 0,Y 149.744,Z 337.834,A -85,B 0,C 180,E1 -24344.894,E2 -24344.894} C_VEL
LIN {X 0,Y 154.809,Z 345.588,A -85,B 0,C 180,E1 -24347.229,E2 -24347.229} C_VEL
LIN {X 0,Y 157.947,Z 350.962,A -85,B 0,C 180,E1 -24348.594,E2 -24348.594} C_VEL
LIN {X 0,Y 163.144,Z 362.714,A -85,B 0,C 180,E1 -24350.843,E2 -24350.843} C_VEL
LIN {X 0,Y 166.646,Z 372.589,A -85,B 0,C 180,E1 -24352.346,E2 -24352.346} C_VEL
LIN {X 0,Y 165.105,Z 400.549,A -85,B 0,C 180,E1 -24353.527,E2 -24353.527} C_VEL
LIN {X 0,Y 163.865,Z 411.042,A -85,B 0,C 180,E1 -24354.261,E2 -24354.261} C_VEL
LIN {X 0,Y 161.768,Z 423.038,A -85,B 0,C 180,E1 -24355.614,E2 -24355.614} C_VEL
LIN {X 0,Y 159.656,Z 432.183,A -85,B 0,C 180,E1 -24357.081,E2 -24357.081} C_VEL
LIN {X 0,Y 157.361,Z 440.217,A -85,B 0,C 180,E1 -24358.723,E2 -24358.723} C_VEL
LIN {X 0,Y 155.085,Z 447.113,A -85,B 0,C 180,E1 -24360.474,E2 -24360.474} C_VEL
LIN {X 0,Y 152.68,Z 453.819,A -85,B 0,C 180,E1 -24362.594,E2 -24362.594} C_VEL
LIN {X 0,Y 150.113,Z 460.171,A -85,B 0,C 180,E1 -24365.08,E2 -24365.08} C_VEL
LIN {X 0,Y 147.799,Z 465.452,A -85,B 0,C 180,E1 -24367.642,E2 -24367.642} C_VEL
LIN {X 0,Y 145.907,Z 469.862,A -85,B 0,C 180,E1 -24370.296,E2 -24370.296} C_VEL
LIN {X 0,Y 143.571,Z 475.051,A -85,B 0,C 180,E1 -24374.382,E2 -24374.382} C_VEL
LIN {X 0,Y 142.414,Z 477.711,A -85,B 0,C 180,E1 -24377.17,E2 -24377.17} C_VEL
LIN {X 0,Y 141.168,Z 480.626,A -85,B 0,C 180,E1 -24381.411,E2 -24381.411} C_VEL
LIN {X 0,Y 140.729,Z 481.896,A -85,B 0,C 180,E1 -24384.268,E2 -24384.268} C_VEL
LIN {X 0,Y 140.538,Z 482.695,A -85,B 0,C 180,E1 -24387.134,E2 -24387.134} C_VEL
LIN {X 0,Y 140.503,Z 482.999,A -85,B 0,C 180,E1 -24390,E2 -24390} C_VEL
LIN {X 0,Y 140.538,Z 482.716,A -85,B 0,C 180,E1 -24392.866,E2 -24392.866} C_VEL
LIN {X 0,Y 140.729,Z 481.96,A -85,B 0,C 180,E1 -24395.732,E2 -24395.732} C_VEL
LIN {X 0,Y 141.167,Z 480.733,A -85,B 0,C 180,E1 -24398.589,E2 -24398.589} C_VEL
LIN {X 0,Y 142.39,Z 477.862,A -85,B 0,C 180,E1 -24402.833,E2 -24402.833} C_VEL
LIN {X 0,Y 143.515,Z 475.248,A -85,B 0,C 180,E1 -24405.624,E2 -24405.624} C_VEL
LIN {X 0,Y 145.862,Z 470.113,A -85,B 0,C 180,E1 -24409.711,E2 -24409.711} C_VEL
LIN {X 0,Y 148.333,Z 464.59,A -85,B 0,C 180,E1 -24413.009,E2 -24413.009} C_VEL
LIN {X 0,Y 151.273,Z 457.646,A -85,B 0,C 180,E1 -24416.19,E2 -24416.19} C_VEL
LIN {X 0,Y 154.328,Z 449.676,A -85,B 0,C 180,E1 -24418.937,E2 -24418.937} C_VEL
LIN {X 0,Y 156.903,Z 442.079,A -85,B 0,C 180,E1 -24421.004,E2 -24421.004} C_VEL
LIN {X 0,Y 159.265,Z 434.085,A -85,B 0,C 180,E1 -24422.728,E2 -24422.728} C_VEL
LIN {X 0,Y 161.144,Z 426.784,A -85,B 0,C 180,E1 -24423.977,E2 -24423.977} C_VEL
LIN {X 0,Y 163.013,Z 416.975,A -85,B 0,C 180,E1 -24425.297,E2 -24425.297} C_VEL
LIN {X 0,Y 164.526,Z 407.297,A -85,B 0,C 180,E1 -24426.194,E2 -24426.194} C_VEL
LIN {X 0,Y 165.51,Z 396.594,A -85,B 0,C 180,E1 -24426.854,E2 -24426.854} C_VEL
LIN {X 0,Y 166.801,Z 373.165,A -85,B 0,C 180,E1 -24427.779,E2 -24427.779} C_VEL
LIN {X 0,Y 165.844,Z 369.766,A -85,B 0,C 180,E1 -24428.218,E2 -24428.218} C_VEL
LIN {X 0,Y 161.075,Z 357.602,A -85,B 0,C 180,E1 -24430.258,E2 -24430.258} C_VEL
LIN {X 0,Y 156.493,Z 348.117,A -85,B 0,C 180,E1 -24432.266,E2 -24432.266} C_VEL
LIN {X 0,Y 150.633,Z 339.184,A -85,B 0,C 180,E1 -24434.91,E2 -24434.91} C_VEL
LIN {X 0,Y 148.752,Z 336.451,A -85,B 0,C 180,E1 -24435.822,E2 -24435.822} C_VEL
LIN {X 0,Y 146.607,Z 333.283,A -85,B 0,C 180,E1 -24436.912,E2 -24436.912} C_VEL
LIN {X 0,Y 145.87,Z 332.266,A -85,B 0,C 180,E1 -24437.295,E2 -24437.295} C_VEL
LIN {X 0,Y 143.904,Z 329.971,A -85,B 0,C 180,E1 -24438.318,E2 -24438.318} C_VEL
LIN {X 0,Y 143.178,Z 327.916,A -85,B 0,C 180,E1 -24439.049,E2 -24439.049} C_VEL
LIN {X 0,Y 143.048,Z 327.415,A -85,B 0,C 180,E1 -24440.305,E2 -24440.305} C_VEL
LIN {X 0,Y 143.156,Z 327.465,A -85,B 0,C 180,E1 -24446.57,E2 -24446.57} C_VEL
LIN {X 0,Y 143.173,Z 327.446,A -85,B 0,C 180,E1 -24452.074,E2 -24452.074} C_VEL
LIN {X 0,Y 143.218,Z 327.43,A -85,B 0,C 180,E1 -24458.804,E2 -24458.804} C_VEL
LIN {X 0,Y 143.247,Z 327.449,A -85,B 0,C 180,E1 -24462.88,E2 -24462.88} C_VEL
LIN {X 0,Y 143.529,Z 327.4,A -85,B 0,C 180,E1 -24468.705,E2 -24468.705} C_VEL
LIN {X 0,Y 143.615,Z 327.404,A -85,B 0,C 180,E1 -24471.558,E2 -24471.558} C_VEL
LIN {X 0,Y 144.148,Z 327.343,A -85,B 0,C 180,E1 -24480,E2 -24480} C_VEL
LIN {X 0,Y 143.599,Z 327.405,A -85,B 0,C 180,E1 -24488.443,E2 -24488.443} C_VEL
LIN {X 0,Y 143.493,Z 327.401,A -85,B 0,C 180,E1 -24491.611,E2 -24491.611} C_VEL
LIN {X 0,Y 143.247,Z 327.448,A -85,B 0,C 180,E1 -24497.12,E2 -24497.12} C_VEL
LIN {X 0,Y 143.217,Z 327.43,A -85,B 0,C 180,E1 -24501.195,E2 -24501.195} C_VEL
LIN {X 0,Y 143.173,Z 327.447,A -85,B 0,C 180,E1 -24507.926,E2 -24507.926} C_VEL
LIN {X 0,Y 143.156,Z 327.465,A -85,B 0,C 180,E1 -24513.429,E2 -24513.429} C_VEL
LIN {X 0,Y 143.048,Z 327.425,A -85,B 0,C 180,E1 -24519.694,E2 -24519.694} C_VEL
LIN {X 0,Y 143.177,Z 327.862,A -85,B 0,C 180,E1 -24520.95,E2 -24520.95} C_VEL
LIN {X 0,Y 143.689,Z 329.511,A -85,B 0,C 180,E1 -24521.593,E2 -24521.593} C_VEL
LIN {X 0,Y 145.315,Z 331.783,A -85,B 0,C 180,E1 -24522.478,E2 -24522.478} C_VEL
LIN {X 0,Y 146.46,Z 332.988,A -85,B 0,C 180,E1 -24523.05,E2 -24523.05} C_VEL
